LIN {X 0,Y 338.282,Z 949.56,A -85,B 0,C 180,E1 15953.701,E2 15953.701} C_VEL
LIN {X 0,Y 337.942,Z 950.503,A -85,B 0,C 180,E1 15950.977,E2 15950.977} C_VEL
LIN {X 0,Y 337.887,Z 949.725,A -85,B 0,C 180,E1 15948.28,E2 15948.28} C_VEL
LIN {X 0,Y 338.122,Z 946.903,A -85,B 0,C 180,E1 15945.416,E2 15945.416} C_VEL
LIN {X 0,Y 338.612,Z 942.779,A -85,B 0,C 180,E1 15942.968,E2 15942.968} C_VEL
LIN {X 0,Y 339.493,Z 936.406,A -85,B 0,C 180,E1 15940.349,E2 15940.349} C_VEL
LIN {X 0,Y 340.591,Z 928.995,A -85,B 0,C 180,E1 15938.1,E2 15938.1} C_VEL
LIN {X 0,Y 342.028,Z 919.535,A -85,B 0,C 180,E1 15935.872,E2 15935.872} C_VEL
LIN {X 0,Y 343.629,Z 908.396,A -85,B 0,C 180,E1 15933.837,E2 15933.837} C_VEL
LIN {X 0,Y 345.191,Z 896.567,A -85,B 0,C 180,E1 15932.124,E2 15932.124} C_VEL
LIN {X 0,Y 346.824,Z 882.835,A -85,B 0,C 180,E1 15930.578,E2 15930.578} C_VEL
LIN {X 0,Y 348.128,Z 869.607,A -85,B 0,C 180,E1 15929.424,E2 15929.424} C_VEL
LIN {X 0,Y 349.323,Z 853.76,A -85,B 0,C 180,E1 15928.401,E2 15928.401} C_VEL
LIN {X 0,Y 350.092,Z 837.915,A -85,B 0,C 180,E1 15927.713,E2 15927.713} C_VEL
LIN {X 0,Y 350.796,Z 811.808,A -85,B 0,C 180,E1 15927.074,E2 15927.074} C_VEL
LIN {X 0,Y 352.568,Z 740.463,A -85,B 0,C 180,E1 15925.552,E2 15925.552} C_VEL
LIN {X 0,Y 347.395,Z 709.374,A -85,B 0,C 180,E1 15924.417,E2 15924.417} C_VEL
LIN {X 0,Y 346.559,Z 706.204,A -85,B 0,C 180,E1 15924.151,E2 15924.151} C_VEL
LIN {X 0,Y 344.566,Z 701.019,A -85,B 0,C 180,E1 15923.183,E2 15923.183} C_VEL
LIN {X 0,Y 342.465,Z 693.939,A -85,B 0,C 180,E1 15921.676,E2 15921.676} C_VEL
LIN {X 0,Y 342.188,Z 686.245,A -85,B 0,C 180,E1 15920.292,E2 15920.292} C_VEL
LIN {X 0,Y 342.295,Z 685.366,A -85,B 0,C 180,E1 15920.142,E2 15920.142} C_VEL
LIN {X 0,Y 345.109,Z 665.644,A -85,B 0,C 180,E1 15916.768,E2 15916.768} C_VEL
LIN {X 0,Y 340.904,Z 649.05,A -85,B 0,C 180,E1 15913.12,E2 15913.12} C_VEL
LIN {X 0,Y 336.381,Z 633.612,A -85,B 0,C 180,E1 15909.442,E2 15909.442} C_VEL
LIN {X 0,Y 331.798,Z 619.998,A -85,B 0,C 180,E1 15905.935,E2 15905.935} C_VEL
LIN {X 0,Y 330.065,Z 614.784,A -85,B 0,C 180,E1 15904.435,E2 15904.435} C_VEL
LIN {X 0,Y 330.051,Z 614.615,A -85,B 0,C 180,E1 15900.009,E2 15900.009} C_VEL
LIN {X 0,Y 330.048,Z 614.676,A -85,B 0,C 180,E1 15895.703,E2 15895.703} C_VEL
LIN {X 0,Y 330.048,Z 614.671,A -85,B 0,C 180,E1 15891.386,E2 15891.386} C_VEL
LIN {X 0,Y 330.04,Z 614.659,A -85,B 0,C 180,E1 15887.151,E2 15887.151} C_VEL
LIN {X 0,Y 330.036,Z 614.677,A -85,B 0,C 180,E1 15882.848,E2 15882.848} C_VEL
LIN {X 0,Y 330.034,Z 614.681,A -85,B 0,C 180,E1 15878.589,E2 15878.589} C_VEL
LIN {X 0,Y 330.027,Z 614.651,A -85,B 0,C 180,E1 15874.198,E2 15874.198} C_VEL
LIN {X 0,Y 330.032,Z 614.688,A -85,B 0,C 180,E1 15869.792,E2 15869.792} C_VEL
LIN {X 0,Y 330.03,Z 614.644,A -85,B 0,C 180,E1 15865.467,E2 15865.467} C_VEL
LIN {X 0,Y 330.038,Z 614.685,A -85,B 0,C 180,E1 15861.132,E2 15861.132} C_VEL
LIN {X 0,Y 330.041,Z 614.643,A -85,B 0,C 180,E1 15856.727,E2 15856.727} C_VEL
LIN {X 0,Y 330.05,Z 614.68,A -85,B 0,C 180,E1 15852.421,E2 15852.421} C_VEL
LIN {X 0,Y 330.055,Z 614.642,A -85,B 0,C 180,E1 15848.011,E2 15848.011} C_VEL
LIN {X 0,Y 330.039,Z 614.678,A -85,B 0,C 180,E1 15843.648,E2 15843.648} C_VEL
LIN {X 0,Y 330.029,Z 614.653,A -85,B 0,C 180,E1 15839.306,E2 15839.306} C_VEL
LIN {X 0,Y 330.021,Z 614.678,A -85,B 0,C 180,E1 15834.96,E2 15834.96} C_VEL
LIN {X 0,Y 330.02,Z 614.672,A -85,B 0,C 180,E1 15830.76,E2 15830.76} C_VEL
LIN {X 0,Y 330.013,Z 614.663,A -85,B 0,C 180,E1 15826.509,E2 15826.509} C_VEL
LIN {X 0,Y 330.014,Z 614.69,A -85,B 0,C 180,E1 15822.182,E2 15822.182} C_VEL
LIN {X 0,Y 330.004,Z 614.675,A -85,B 0,C 180,E1 15817.933,E2 15817.933} C_VEL
LIN {X 0,Y 330.01,Z 614.666,A -85,B 0,C 180,E1 15813.553,E2 15813.553} C_VEL
LIN {X 0,Y 330.005,Z 614.672,A -85,B 0,C 180,E1 15809.371,E2 15809.371} C_VEL
LIN {X 0,Y 330.008,Z 614.675,A -85,B 0,C 180,E1 15805.194,E2 15805.194} C_VEL
LIN {X 0,Y 330.031,Z 614.845,A -85,B 0,C 180,E1 15800.976,E2 15800.976} C_VEL
LIN {X 0,Y 334.572,Z 626.543,A -85,B 0,C 180,E1 15798.208,E2 15798.208} C_VEL
LIN {X 0,Y 340.383,Z 642.032,A -85,B 0,C 180,E1 15794.934,E2 15794.934} C_VEL
LIN {X 0,Y 346.42,Z 659.693,A -85,B 0,C 180,E1 15791.594,E2 15791.594} C_VEL
LIN {X 0,Y 351.026,Z 674.252,A -85,B 0,C 180,E1 15789.066,E2 15789.066} C_VEL
LIN {X 0,Y 347.702,Z 695.465,A -85,B 0,C 180,E1 15786.551,E2 15786.551} C_VEL
LIN {X 0,Y 350.631,Z 727.811,A -85,B 0,C 180,E1 15785.557,E2 15785.557} C_VEL
LIN {X 0,Y 346.435,Z 886.846,A -85,B 0,C 180,E1 15782.34,E2 15782.34} C_VEL
LIN {X 0,Y 345.21,Z 905.278,A -85,B 0,C 180,E1 15781.685,E2 15781.685} C_VEL
LIN {X 0,Y 343.439,Z 923.152,A -85,B 0,C 180,E1 15780.753,E2 15780.753} C_VEL
LIN {X 0,Y 341.468,Z 939.767,A -85,B 0,C 180,E1 15779.582,E2 15779.582} C_VEL
LIN {X 0,Y 339.185,Z 956.678,A -85,B 0,C 180,E1 15778.046,E2 15778.046} C_VEL
LIN {X 0,Y 336.841,Z 972.419,A -85,B 0,C 180,E1 15776.25,E2 15776.25} C_VEL
LIN {X 0,Y 334.602,Z 987.176,A -85,B 0,C 180,E1 15774.167,E2 15774.167} C_VEL
LIN {X 0,Y 332.635,Z 1000.358,A -85,B 0,C 180,E1 15771.884,E2 15771.884} C_VEL
LIN {X 0,Y 331.024,Z 1012.138,A -85,B 0,C 180,E1 15769.406,E2 15769.406} C_VEL
LIN {X 0,Y 329.802,Z 1022.804,A -85,B 0,C 180,E1 15766.662,E2 15766.662} C_VEL
LIN {X 0,Y 329.096,Z 1032.024,A -85,B 0,C 180,E1 15763.709,E2 15763.709} C_VEL
LIN {X 0,Y 328.87,Z 1039.391,A -85,B 0,C 180,E1 15760.688,E2 15760.688} C_VEL
LIN {X 0,Y 329.024,Z 1044.857,A -85,B 0,C 180,E1 15757.684,E2 15757.684} C_VEL
LIN {X 0,Y 329.333,Z 1048.545,A -85,B 0,C 180,E1 15754.702,E2 15754.702} C_VEL
LIN {X 0,Y 329.583,Z 1050.525,A -85,B 0,C 180,E1 15751.739,E2 15751.739} C_VEL
LIN {X 0,Y 329.594,Z 1050.859,A -85,B 0,C 180,E1 15748.957,E2 15748.957} C_VEL
LIN {X 0,Y 329.364,Z 1049.731,A -85,B 0,C 180,E1 15746.171,E2 15746.171} C_VEL
LIN {X 0,Y 329.013,Z 1046.925,A -85,B 0,C 180,E1 15743.194,E2 15743.194} C_VEL
LIN {X 0,Y 328.773,Z 1042.425,A -85,B 0,C 180,E1 15740.177,E2 15740.177} C_VEL
LIN {X 0,Y 328.894,Z 1035.816,A -85,B 0,C 180,E1 15736.999,E2 15736.999} C_VEL
LIN {X 0,Y 329.539,Z 1027.629,A -85,B 0,C 180,E1 15733.972,E2 15733.972} C_VEL
LIN {X 0,Y 330.842,Z 1017.333,A -85,B 0,C 180,E1 15730.95,E2 15730.95} C_VEL
LIN {X 0,Y 332.674,Z 1005.885,A -85,B 0,C 180,E1 15728.234,E2 15728.234} C_VEL
LIN {X 0,Y 334.846,Z 993.661,A -85,B 0,C 180,E1 15725.853,E2 15725.853} C_VEL
LIN {X 0,Y 337.541,Z 979.122,A -85,B 0,C 180,E1 15723.525,E2 15723.525} C_VEL
LIN {X 0,Y 340.344,Z 964.071,A -85,B 0,C 180,E1 15721.581,E2 15721.581} C_VEL
LIN {X 0,Y 343.092,Z 948.032,A -85,B 0,C 180,E1 15719.917,E2 15719.917} C_VEL
LIN {X 0,Y 345.607,Z 931.814,A -85,B 0,C 180,E1 15718.589,E2 15718.589} C_VEL
LIN {X 0,Y 347.921,Z 914.248,A -85,B 0,C 180,E1 15717.493,E2 15717.493} C_VEL
LIN {X 0,Y 349.839,Z 895.574,A -85,B 0,C 180,E1 15716.67,E2 15716.67} C_VEL
LIN {X 0,Y 350.907,Z 877.121,A -85,B 0,C 180,E1 15716.145,E2 15716.145} C_VEL
LIN {X 0,Y 355.545,Z 725.644,A -85,B 0,C 180,E1 15713.02,E2 15713.02} C_VEL
LIN {X 0,Y 352.544,Z 696.426,A -85,B 0,C 180,E1 15711.908,E2 15711.908} C_VEL
LIN {X 0,Y 355.73,Z 679.777,A -85,B 0,C 180,E1 15709.864,E2 15709.864} C_VEL
LIN {X 0,Y 351.383,Z 665.481,A -85,B 0,C 180,E1 15706.928,E2 15706.928} C_VEL
LIN {X 0,Y 346.624,Z 652.331,A -85,B 0,C 180,E1 15703.812,E2 15703.812} C_VEL
LIN {X 0,Y 341.748,Z 640.208,A -85,B 0,C 180,E1 15700.475,E2 15700.475} C_VEL
LIN {X 0,Y 337.434,Z 630.747,A -85,B 0,C 180,E1 15697.404,E2 15697.404} C_VEL
LIN {X 0,Y 335.51,Z 626.722,A -85,B 0,C 180,E1 15695.95,E2 15695.95} C_VEL
LIN {X 0,Y 333.99,Z 623.294,A -85,B 0,C 180,E1 15694.666,E2 15694.666} C_VEL
LIN {X 0,Y 331.766,Z 618.774,A -85,B 0,C 180,E1 15692.772,E2 15692.772} C_VEL
LIN {X 0,Y 330.033,Z 614.822,A -85,B 0,C 180,E1 15690.923,E2 15690.923} C_VEL
LIN {X 0,Y 330.021,Z 614.671,A -85,B 0,C 180,E1 15686.835,E2 15686.835} C_VEL
LIN {X 0,Y 330.015,Z 614.669,A -85,B 0,C 180,E1 15682.63,E2 15682.63} C_VEL
LIN {X 0,Y 330.015,Z 614.666,A -85,B 0,C 180,E1 15678.366,E2 15678.366} C_VEL
LIN {X 0,Y 330.013,Z 614.663,A -85,B 0,C 180,E1 15674.182,E2 15674.182} C_VEL
LIN {X 0,Y 330.016,Z 614.663,A -85,B 0,C 180,E1 15669.944,E2 15669.944} C_VEL
LIN {X 0,Y 330.011,Z 614.668,A -85,B 0,C 180,E1 15665.563,E2 15665.563} C_VEL
LIN {X 0,Y 330.016,Z 614.674,A -85,B 0,C 180,E1 15661.117,E2 15661.117} C_VEL
LIN {X 0,Y 330.02,Z 614.683,A -85,B 0,C 180,E1 15656.873,E2 15656.873} C_VEL
LIN {X 0,Y 330.03,Z 614.685,A -85,B 0,C 180,E1 15652.514,E2 15652.514} C_VEL
LIN {X 0,Y 330.039,Z 614.681,A -85,B 0,C 180,E1 15648.107,E2 15648.107} C_VEL
LIN {X 0,Y 330.057,Z 614.851,A -85,B 0,C 180,E1 15644.088,E2 15644.088} C_VEL
LIN {X 0,Y 331.806,Z 618.825,A -85,B 0,C 180,E1 15642.099,E2 15642.099} C_VEL
LIN {X 0,Y 334.242,Z 624.749,A -85,B 0,C 180,E1 15639.512,E2 15639.512} C_VEL
LIN {X 0,Y 337.03,Z 631.317,A -85,B 0,C 180,E1 15636.878,E2 15636.878} C_VEL
LIN {X 0,Y 340.661,Z 640.852,A -85,B 0,C 180,E1 15633.504,E2 15633.504} C_VEL
LIN {X 0,Y 344.388,Z 651.989,A -85,B 0,C 180,E1 15630.041,E2 15630.041} C_VEL
LIN {X 0,Y 347.816,Z 664.12,A -85,B 0,C 180,E1 15626.697,E2 15626.697} C_VEL
LIN {X 0,Y 350.134,Z 674.513,A -85,B 0,C 180,E1 15624.117,E2 15624.117} C_VEL
LIN {X 0,Y 345.344,Z 700.754,A -85,B 0,C 180,E1 15619.464,E2 15619.464} C_VEL
LIN {X 0,Y 344.564,Z 706.075,A -85,B 0,C 180,E1 15618.576,E2 15618.576} C_VEL
LIN {X 0,Y 350.106,Z 734.115,A -85,B 0,C 180,E1 15617.096,E2 15617.096} C_VEL
LIN {X 0,Y 351.866,Z 746.069,A -85,B 0,C 180,E1 15616.573,E2 15616.573} C_VEL
LIN {X 0,Y 348.485,Z 837.417,A -85,B 0,C 180,E1 15614.49,E2 15614.49} C_VEL
LIN {X 0,Y 347.514,Z 853.648,A -85,B 0,C 180,E1 15613.812,E2 15613.812} C_VEL
LIN {X 0,Y 346.161,Z 868.356,A -85,B 0,C 180,E1 15612.908,E2 15612.908} C_VEL
LIN {X 0,Y 344.33,Z 882.931,A -85,B 0,C 180,E1 15611.68,E2 15611.68} C_VEL
LIN {X 0,Y 342.265,Z 896.285,A -85,B 0,C 180,E1 15610.211,E2 15610.211} C_VEL
LIN {X 0,Y 339.904,Z 909.258,A -85,B 0,C 180,E1 15608.365,E2 15608.365} C_VEL
LIN {X 0,Y 337.831,Z 919.497,A -85,B 0,C 180,E1 15606.504,E2 15606.504} C_VEL
LIN {X 0,Y 335.671,Z 929.228,A -85,B 0,C 180,E1 15604.261,E2 15604.261} C_VEL
LIN {X 0,Y 333.889,Z 936.762,A -85,B 0,C 180,E1 15602.008,E2 15602.008} C_VEL
LIN {X 0,Y 332.297,Z 943.342,A -85,B 0,C 180,E1 15599.37,E2 15599.37} C_VEL
LIN {X 0,Y 331.171,Z 947.855,A -85,B 0,C 180,E1 15596.734,E2 15596.734} C_VEL
LIN {X 0,Y 330.426,Z 950.744,A -85,B 0,C 180,E1 15593.921,E2 15593.921} C_VEL
LIN {X 0,Y 330.041,Z 951.708,A -85,B 0,C 180,E1 15591.078,E2 15591.078} C_VEL
LIN {X 0,Y 329.972,Z 950.962,A -85,B 0,C 180,E1 15588.369,E2 15588.369} C_VEL
LIN {X 0,Y 330.176,Z 948.422,A -85,B 0,C 180,E1 15585.635,E2 15585.635} C_VEL
LIN {X 0,Y 330.709,Z 944.112,A -85,B 0,C 180,E1 15582.928,E2 15582.928} C_VEL
LIN {X 0,Y 331.617,Z 937.787,A -85,B 0,C 180,E1 15580.247,E2 15580.247} C_VEL
LIN {X 0,Y 332.755,Z 930.471,A -85,B 0,C 180,E1 15577.945,E2 15577.945} C_VEL
LIN {X 0,Y 334.239,Z 921.09,A -85,B 0,C 180,E1 15575.665,E2 15575.665} C_VEL
LIN {X 0,Y 335.828,Z 910.621,A -85,B 0,C 180,E1 15573.67,E2 15573.67} C_VEL
LIN {X 0,Y 337.533,Z 898.355,A -85,B 0,C 180,E1 15571.819,E2 15571.819} C_VEL
LIN {X 0,Y 339.205,Z 884.971,A -85,B 0,C 180,E1 15570.253,E2 15570.253} C_VEL
LIN {X 0,Y 340.661,Z 871.088,A -85,B 0,C 180,E1 15568.991,E2 15568.991} C_VEL
LIN {X 0,Y 341.902,Z 855.452,A -85,B 0,C 180,E1 15567.947,E2 15567.947} C_VEL
LIN {X 0,Y 342.73,Z 839.818,A -85,B 0,C 180,E1 15567.23,E2 15567.23} C_VEL
LIN {X 0,Y 343.359,Z 817.533,A -85,B 0,C 180,E1 15566.648,E2 15566.648} C_VEL
LIN {X 0,Y 345.371,Z 741.623,A -85,B 0,C 180,E1 15564.998,E2 15564.998} C_VEL
LIN {X 0,Y 339.605,Z 706.444,A -85,B 0,C 180,E1 15563.661,E2 15563.661} C_VEL
LIN {X 0,Y 341.799,Z 688.88,A -85,B 0,C 180,E1 15560.741,E2 15560.741} C_VEL
LIN {X 0,Y 342.295,Z 685.366,A -85,B 0,C 180,E1 15560.142,E2 15560.142} C_VEL
LIN {X 0,Y 342.241,Z 680.167,A -85,B 0,C 180,E1 15559.178,E2 15559.178} C_VEL
LIN {X 0,Y 340.277,Z 673.413,A -85,B 0,C 180,E1 15557.717,E2 15557.717} C_VEL
LIN {X 0,Y 336.594,Z 663.57,A -85,B 0,C 180,E1 15555.441,E2 15555.441} C_VEL
LIN {X 0,Y 332.394,Z 647.593,A -85,B 0,C 180,E1 15551.769,E2 15551.769} C_VEL
LIN {X 0,Y 328.021,Z 633.059,A -85,B 0,C 180,E1 15548.168,E2 15548.168} C_VEL
LIN {X 0,Y 323.24,Z 618.973,A -85,B 0,C 180,E1 15544.338,E2 15544.338} C_VEL
LIN {X 0,Y 322.115,Z 615.767,A -85,B 0,C 180,E1 15543.305,E2 15543.305} C_VEL
LIN {X 0,Y 322.094,Z 615.599,A -85,B 0,C 180,E1 15538.957,E2 15538.957} C_VEL
LIN {X 0,Y 322.107,Z 615.676,A -85,B 0,C 180,E1 15534.516,E2 15534.516} C_VEL
LIN {X 0,Y 322.119,Z 615.677,A -85,B 0,C 180,E1 15530.019,E2 15530.019} C_VEL
LIN {X 0,Y 322.111,Z 615.657,A -85,B 0,C 180,E1 15525.557,E2 15525.557} C_VEL
LIN {X 0,Y 322.113,Z 615.639,A -85,B 0,C 180,E1 15521.153,E2 15521.153} C_VEL
LIN {X 0,Y 322.103,Z 615.673,A -85,B 0,C 180,E1 15516.786,E2 15516.786} C_VEL
LIN {X 0,Y 322.093,Z 615.649,A -85,B 0,C 180,E1 15512.396,E2 15512.396} C_VEL
LIN {X 0,Y 322.093,Z 615.659,A -85,B 0,C 180,E1 15508.155,E2 15508.155} C_VEL
LIN {X 0,Y 322.086,Z 615.662,A -85,B 0,C 180,E1 15503.682,E2 15503.682} C_VEL
LIN {X 0,Y 322.085,Z 615.647,A -85,B 0,C 180,E1 15499.313,E2 15499.313} C_VEL
LIN {X 0,Y 322.093,Z 615.661,A -85,B 0,C 180,E1 15494.931,E2 15494.931} C_VEL
LIN {X 0,Y 322.098,Z 615.644,A -85,B 0,C 180,E1 15490.554,E2 15490.554} C_VEL
LIN {X 0,Y 322.11,Z 615.658,A -85,B 0,C 180,E1 15486.237,E2 15486.237} C_VEL
LIN {X 0,Y 322.106,Z 615.637,A -85,B 0,C 180,E1 15481.735,E2 15481.735} C_VEL
LIN {X 0,Y 322.105,Z 615.67,A -85,B 0,C 180,E1 15477.51,E2 15477.51} C_VEL
LIN {X 0,Y 322.099,Z 615.636,A -85,B 0,C 180,E1 15473.226,E2 15473.226} C_VEL
LIN {X 0,Y 322.087,Z 615.677,A -85,B 0,C 180,E1 15468.806,E2 15468.806} C_VEL
LIN {X 0,Y 322.078,Z 615.652,A -85,B 0,C 180,E1 15464.516,E2 15464.516} C_VEL
LIN {X 0,Y 322.074,Z 615.655,A -85,B 0,C 180,E1 15460.162,E2 15460.162} C_VEL
LIN {X 0,Y 322.072,Z 615.676,A -85,B 0,C 180,E1 15455.809,E2 15455.809} C_VEL
LIN {X 0,Y 322.075,Z 615.68,A -85,B 0,C 180,E1 15451.44,E2 15451.44} C_VEL
LIN {X 0,Y 322.081,Z 615.679,A -85,B 0,C 180,E1 15447.094,E2 15447.094} C_VEL
LIN {X 0,Y 322.087,Z 615.675,A -85,B 0,C 180,E1 15442.747,E2 15442.747} C_VEL
LIN {X 0,Y 322.162,Z 616.103,A -85,B 0,C 180,E1 15442.008,E2 15442.008} C_VEL
LIN {X 0,Y 327.813,Z 630.366,A -85,B 0,C 180,E1 15438.558,E2 15438.558} C_VEL
LIN {X 0,Y 333.879,Z 646.764,A -85,B 0,C 180,E1 15435.03,E2 15435.03} C_VEL
LIN {X 0,Y 339.979,Z 664.942,A -85,B 0,C 180,E1 15431.542,E2 15431.542} C_VEL
LIN {X 0,Y 343.602,Z 676.825,A -85,B 0,C 180,E1 15429.449,E2 15429.449} C_VEL
LIN {X 0,Y 340.552,Z 695.511,A -85,B 0,C 180,E1 15427.185,E2 15427.185} C_VEL
LIN {X 0,Y 343.459,Z 728.591,A -85,B 0,C 180,E1 15426.135,E2 15426.135} C_VEL
LIN {X 0,Y 339.118,Z 886.31,A -85,B 0,C 180,E1 15422.886,E2 15422.886} C_VEL
LIN {X 0,Y 337.856,Z 904.729,A -85,B 0,C 180,E1 15422.22,E2 15422.22} C_VEL
LIN {X 0,Y 336.011,Z 922.754,A -85,B 0,C 180,E1 15421.26,E2 15421.26} C_VEL
LIN {X 0,Y 333.876,Z 940.037,A -85,B 0,C 180,E1 15420.008,E2 15420.008} C_VEL
LIN {X 0,Y 331.546,Z 956.6,A -85,B 0,C 180,E1 15418.457,E2 15418.457} C_VEL
LIN {X 0,Y 329.135,Z 972.132,A -85,B 0,C 180,E1 15416.63,E2 15416.63} C_VEL
LIN {X 0,Y 326.805,Z 986.777,A -85,B 0,C 180,E1 15414.492,E2 15414.492} C_VEL
LIN {X 0,Y 324.704,Z 1000.299,A -85,B 0,C 180,E1 15412.066,E2 15412.066} C_VEL
LIN {X 0,Y 323.057,Z 1011.911,A -85,B 0,C 180,E1 15409.528,E2 15409.528} C_VEL
LIN {X 0,Y 321.782,Z 1022.775,A -85,B 0,C 180,E1 15406.611,E2 15406.611} C_VEL
LIN {X 0,Y 321.114,Z 1031.499,A -85,B 0,C 180,E1 15403.689,E2 15403.689} C_VEL
LIN {X 0,Y 320.91,Z 1038.731,A -85,B 0,C 180,E1 15400.593,E2 15400.593} C_VEL
LIN {X 0,Y 321.098,Z 1044.066,A -85,B 0,C 180,E1 15397.515,E2 15397.515} C_VEL
LIN {X 0,Y 321.418,Z 1047.441,A -85,B 0,C 180,E1 15394.64,E2 15394.64} C_VEL
LIN {X 0,Y 321.671,Z 1049.298,A -85,B 0,C 180,E1 15391.782,E2 15391.782} C_VEL
LIN {X 0,Y 321.681,Z 1049.666,A -85,B 0,C 180,E1 15388.932,E2 15388.932} C_VEL
LIN {X 0,Y 321.423,Z 1048.563,A -85,B 0,C 180,E1 15386.076,E2 15386.076} C_VEL
LIN {X 0,Y 321.042,Z 1045.778,A -85,B 0,C 180,E1 15383.024,E2 15383.024} C_VEL
LIN {X 0,Y 320.792,Z 1041.326,A -85,B 0,C 180,E1 15379.948,E2 15379.948} C_VEL
LIN {X 0,Y 320.946,Z 1034.696,A -85,B 0,C 180,E1 15376.672,E2 15376.672} C_VEL
LIN {X 0,Y 321.656,Z 1026.519,A -85,B 0,C 180,E1 15373.569,E2 15373.569} C_VEL
LIN {X 0,Y 322.971,Z 1016.901,A -85,B 0,C 180,E1 15370.655,E2 15370.655} C_VEL
LIN {X 0,Y 324.984,Z 1005.117,A -85,B 0,C 180,E1 15367.764,E2 15367.764} C_VEL
LIN {X 0,Y 327.361,Z 992.635,A -85,B 0,C 180,E1 15365.264,E2 15365.264} C_VEL
LIN {X 0,Y 330.105,Z 978.696,A -85,B 0,C 180,E1 15362.978,E2 15362.978} C_VEL
LIN {X 0,Y 333.036,Z 963.853,A -85,B 0,C 180,E1 15361.003,E2 15361.003} C_VEL
LIN {X 0,Y 335.906,Z 948.039,A -85,B 0,C 180,E1 15359.314,E2 15359.314} C_VEL
LIN {X 0,Y 338.66,Z 931.126,A -85,B 0,C 180,E1 15357.898,E2 15357.898} C_VEL
LIN {X 0,Y 341.043,Z 913.911,A -85,B 0,C 180,E1 15356.804,E2 15356.804} C_VEL
LIN {X 0,Y 343.046,Z 895.285,A -85,B 0,C 180,E1 15355.965,E2 15355.965} C_VEL
LIN {X 0,Y 344.178,Z 876.781,A -85,B 0,C 180,E1 15355.425,E2 15355.425} C_VEL
LIN {X 0,Y 349.065,Z 726.518,A -85,B 0,C 180,E1 15352.264,E2 15352.264} C_VEL
LIN {X 0,Y 346.022,Z 696.479,A -85,B 0,C 180,E1 15351.079,E2 15351.079} C_VEL
LIN {X 0,Y 348.734,Z 682.628,A -85,B 0,C 180,E1 15349.331,E2 15349.331} C_VEL
LIN {X 0,Y 344.703,Z 669.207,A -85,B 0,C 180,E1 15346.482,E2 15346.482} C_VEL
LIN {X 0,Y 339.842,Z 655.593,A -85,B 0,C 180,E1 15343.143,E2 15343.143} C_VEL
LIN {X 0,Y 335.228,Z 644.252,A -85,B 0,C 180,E1 15339.886,E2 15339.886} C_VEL
LIN {X 0,Y 330.696,Z 633.649,A -85,B 0,C 180,E1 15336.342,E2 15336.342} C_VEL
LIN {X 0,Y 327.861,Z 628.133,A -85,B 0,C 180,E1 15334.134,E2 15334.134} C_VEL
LIN {X 0,Y 326.265,Z 624.54,A -85,B 0,C 180,E1 15332.64,E2 15332.64} C_VEL
LIN {X 0,Y 323.893,Z 619.847,A -85,B 0,C 180,E1 15330.415,E2 15330.415} C_VEL
LIN {X 0,Y 322.088,Z 615.8,A -85,B 0,C 180,E1 15328.2,E2 15328.2} C_VEL
LIN {X 0,Y 322.076,Z 615.654,A -85,B 0,C 180,E1 15323.801,E2 15323.801} C_VEL
LIN {X 0,Y 322.08,Z 615.654,A -85,B 0,C 180,E1 15319.589,E2 15319.589} C_VEL
LIN {X 0,Y 322.087,Z 615.656,A -85,B 0,C 180,E1 15315.299,E2 15315.299} C_VEL
LIN {X 0,Y 322.098,Z 615.66,A -85,B 0,C 180,E1 15310.915,E2 15310.915} C_VEL
LIN {X 0,Y 322.117,Z 615.669,A -85,B 0,C 180,E1 15306.595,E2 15306.595} C_VEL
LIN {X 0,Y 322.102,Z 615.677,A -85,B 0,C 180,E1 15302.134,E2 15302.134} C_VEL
LIN {X 0,Y 322.099,Z 615.67,A -85,B 0,C 180,E1 15297.865,E2 15297.865} C_VEL
LIN {X 0,Y 322.088,Z 615.668,A -85,B 0,C 180,E1 15293.402,E2 15293.402} C_VEL
LIN {X 0,Y 322.086,Z 615.668,A -85,B 0,C 180,E1 15289.084,E2 15289.084} C_VEL
LIN {X 0,Y 322.132,Z 616.005,A -85,B 0,C 180,E1 15286.63,E2 15286.63} C_VEL
LIN {X 0,Y 324.448,Z 621.314,A -85,B 0,C 180,E1 15283.713,E2 15283.713} C_VEL
LIN {X 0,Y 326.371,Z 625.626,A -85,B 0,C 180,E1 15281.606,E2 15281.606} C_VEL
LIN {X 0,Y 328.211,Z 629.924,A -85,B 0,C 180,E1 15279.678,E2 15279.678} C_VEL
LIN {X 0,Y 331.031,Z 636.814,A -85,B 0,C 180,E1 15276.88,E2 15276.88} C_VEL
LIN {X 0,Y 334.3,Z 645.526,A -85,B 0,C 180,E1 15273.726,E2 15273.726} C_VEL
LIN {X 0,Y 337.901,Z 656.63,A -85,B 0,C 180,E1 15270.19,E2 15270.19} C_VEL
LIN {X 0,Y 341.08,Z 668.141,A -85,B 0,C 180,E1 15266.958,E2 15266.958} C_VEL
LIN {X 0,Y 343.152,Z 677.532,A -85,B 0,C 180,E1 15264.56,E2 15264.56} C_VEL
LIN {X 0,Y 338.173,Z 703.553,A -85,B 0,C 180,E1 15259.868,E2 15259.868} C_VEL
LIN {X 0,Y 337.894,Z 706.302,A -85,B 0,C 180,E1 15259.451,E2 15259.451} C_VEL
LIN {X 0,Y 343.67,Z 735.552,A -85,B 0,C 180,E1 15257.866,E2 15257.866} C_VEL
LIN {X 0,Y 345.402,Z 747.206,A -85,B 0,C 180,E1 15257.334,E2 15257.334} C_VEL
LIN {X 0,Y 341.868,Z 838.036,A -85,B 0,C 180,E1 15255.23,E2 15255.23} C_VEL
LIN {X 0,Y 340.84,Z 854.294,A -85,B 0,C 180,E1 15254.54,E2 15254.54} C_VEL
LIN {X 0,Y 339.356,Z 869.483,A -85,B 0,C 180,E1 15253.586,E2 15253.586} C_VEL
LIN {X 0,Y 337.349,Z 884.526,A -85,B 0,C 180,E1 15252.283,E2 15252.283} C_VEL
LIN {X 0,Y 335.172,Z 897.677,A -85,B 0,C 180,E1 15250.791,E2 15250.791} C_VEL
LIN {X 0,Y 332.687,Z 910.556,A -85,B 0,C 180,E1 15248.912,E2 15248.912} C_VEL
LIN {X 0,Y 330.291,Z 921.628,A -85,B 0,C 180,E1 15246.826,E2 15246.826} C_VEL
LIN {X 0,Y 328.04,Z 931.147,A -85,B 0,C 180,E1 15244.536,E2 15244.536} C_VEL
LIN {X 0,Y 326.036,Z 939.016,A -85,B 0,C 180,E1 15242.042,E2 15242.042} C_VEL
LIN {X 0,Y 324.506,Z 944.917,A -85,B 0,C 180,E1 15239.537,E2 15239.537} C_VEL
LIN {X 0,Y 323.247,Z 949.563,A -85,B 0,C 180,E1 15236.628,E2 15236.628} C_VEL
LIN {X 0,Y 322.511,Z 952.107,A -85,B 0,C 180,E1 15233.854,E2 15233.854} C_VEL
LIN {X 0,Y 322.119,Z 952.926,A -85,B 0,C 180,E1 15230.882,E2 15230.882} C_VEL
LIN {X 0,Y 322.062,Z 951.937,A -85,B 0,C 180,E1 15228.086,E2 15228.086} C_VEL
LIN {X 0,Y 322.313,Z 949.186,A -85,B 0,C 180,E1 15225.253,E2 15225.253} C_VEL
LIN {X 0,Y 322.898,Z 944.675,A -85,B 0,C 180,E1 15222.518,E2 15222.518} C_VEL
LIN {X 0,Y 323.822,Z 938.62,A -85,B 0,C 180,E1 15219.943,E2 15219.943} C_VEL
LIN {X 0,Y 325.019,Z 931.247,A -85,B 0,C 180,E1 15217.601,E2 15217.601} C_VEL
LIN {X 0,Y 326.583,Z 921.799,A -85,B 0,C 180,E1 15215.27,E2 15215.27} C_VEL
LIN {X 0,Y 328.327,Z 910.715,A -85,B 0,C 180,E1 15213.142,E2 15213.142} C_VEL
LIN {X 0,Y 330.046,Z 898.834,A -85,B 0,C 180,E1 15211.333,E2 15211.333} C_VEL
LIN {X 0,Y 331.787,Z 885.386,A -85,B 0,C 180,E1 15209.741,E2 15209.741} C_VEL
LIN {X 0,Y 333.304,Z 871.356,A -85,B 0,C 180,E1 15208.453,E2 15208.453} C_VEL
LIN {X 0,Y 334.6,Z 855.565,A -85,B 0,C 180,E1 15207.388,E2 15207.388} C_VEL
LIN {X 0,Y 335.447,Z 839.861,A -85,B 0,C 180,E1 15206.668,E2 15206.668} C_VEL
LIN {X 0,Y 336.137,Z 816.358,A -85,B 0,C 180,E1 15206.053,E2 15206.053} C_VEL
LIN {X 0,Y 338.188,Z 742.721,A -85,B 0,C 180,E1 15204.422,E2 15204.422} C_VEL
LIN {X 0,Y 332.289,Z 706.332,A -85,B 0,C 180,E1 15203,E2 15203} C_VEL
LIN {X 0,Y 333.364,Z 697.56,A -85,B 0,C 180,E1 15201.548,E2 15201.548} C_VEL
LIN {X 0,Y 337.399,Z 670.235,A -85,B 0,C 180,E1 15196.809,E2 15196.809} C_VEL
LIN {X 0,Y 337.527,Z 667.454,A -85,B 0,C 180,E1 15196.291,E2 15196.291} C_VEL
LIN {X 0,Y 336.594,Z 663.57,A -85,B 0,C 180,E1 15195.441,E2 15195.441} C_VEL
LIN {X 0,Y 334.538,Z 659.376,A -85,B 0,C 180,E1 15194.383,E2 15194.383} C_VEL
LIN {X 0,Y 325.4,Z 649.582,A -85,B 0,C 180,E1 15191.255,E2 15191.255} C_VEL
LIN {X 0,Y 324.049,Z 646.601,A -85,B 0,C 180,E1 15190.454,E2 15190.454} C_VEL
LIN {X 0,Y 319.525,Z 632.114,A -85,B 0,C 180,E1 15186.681,E2 15186.681} C_VEL
LIN {X 0,Y 315.121,Z 619.584,A -85,B 0,C 180,E1 15183.075,E2 15183.075} C_VEL
LIN {X 0,Y 314.193,Z 616.761,A -85,B 0,C 180,E1 15182.165,E2 15182.165} C_VEL
LIN {X 0,Y 314.164,Z 616.594,A -85,B 0,C 180,E1 15177.842,E2 15177.842} C_VEL
LIN {X 0,Y 314.166,Z 616.649,A -85,B 0,C 180,E1 15173.476,E2 15173.476} C_VEL
LIN {X 0,Y 314.162,Z 616.658,A -85,B 0,C 180,E1 15168.963,E2 15168.963} C_VEL
LIN {X 0,Y 314.161,Z 616.663,A -85,B 0,C 180,E1 15164.442,E2 15164.442} C_VEL
LIN {X 0,Y 314.166,Z 616.632,A -85,B 0,C 180,E1 15159.914,E2 15159.914} C_VEL
LIN {X 0,Y 314.169,Z 616.64,A -85,B 0,C 180,E1 15155.438,E2 15155.438} C_VEL
LIN {X 0,Y 314.181,Z 616.655,A -85,B 0,C 180,E1 15151.035,E2 15151.035} C_VEL
LIN {X 0,Y 314.166,Z 616.62,A -85,B 0,C 180,E1 15146.579,E2 15146.579} C_VEL
LIN {X 0,Y 314.156,Z 616.663,A -85,B 0,C 180,E1 15142.059,E2 15142.059} C_VEL
LIN {X 0,Y 314.142,Z 616.617,A -85,B 0,C 180,E1 15137.6,E2 15137.6} C_VEL
LIN {X 0,Y 314.147,Z 616.666,A -85,B 0,C 180,E1 15133.109,E2 15133.109} C_VEL
LIN {X 0,Y 314.152,Z 616.616,A -85,B 0,C 180,E1 15128.603,E2 15128.603} C_VEL
LIN {X 0,Y 314.163,Z 616.66,A -85,B 0,C 180,E1 15124.198,E2 15124.198} C_VEL
LIN {X 0,Y 314.173,Z 616.621,A -85,B 0,C 180,E1 15119.636,E2 15119.636} C_VEL
LIN {X 0,Y 314.158,Z 616.657,A -85,B 0,C 180,E1 15115.254,E2 15115.254} C_VEL
LIN {X 0,Y 314.146,Z 616.644,A -85,B 0,C 180,E1 15110.843,E2 15110.843} C_VEL
LIN {X 0,Y 314.131,Z 616.638,A -85,B 0,C 180,E1 15106.377,E2 15106.377} C_VEL
LIN {X 0,Y 314.138,Z 616.667,A -85,B 0,C 180,E1 15101.825,E2 15101.825} C_VEL
LIN {X 0,Y 314.135,Z 616.656,A -85,B 0,C 180,E1 15097.546,E2 15097.546} C_VEL
LIN {X 0,Y 314.151,Z 616.643,A -85,B 0,C 180,E1 15093.132,E2 15093.132} C_VEL
LIN {X 0,Y 314.165,Z 616.644,A -85,B 0,C 180,E1 15088.751,E2 15088.751} C_VEL
LIN {X 0,Y 314.161,Z 616.651,A -85,B 0,C 180,E1 15084.251,E2 15084.251} C_VEL
LIN {X 0,Y 314.191,Z 617.076,A -85,B 0,C 180,E1 15083.229,E2 15083.229} C_VEL
LIN {X 0,Y 319.821,Z 630.963,A -85,B 0,C 180,E1 15079.674,E2 15079.674} C_VEL
LIN {X 0,Y 325.933,Z 647.385,A -85,B 0,C 180,E1 15075.987,E2 15075.987} C_VEL
LIN {X 0,Y 331.742,Z 664.66,A -85,B 0,C 180,E1 15072.518,E2 15072.518} C_VEL
LIN {X 0,Y 336.242,Z 679.007,A -85,B 0,C 180,E1 15069.897,E2 15069.897} C_VEL
LIN {X 0,Y 333.42,Z 695.85,A -85,B 0,C 180,E1 15067.82,E2 15067.82} C_VEL
LIN {X 0,Y 336.325,Z 729.344,A -85,B 0,C 180,E1 15066.738,E2 15066.738} C_VEL
LIN {X 0,Y 331.822,Z 885.719,A -85,B 0,C 180,E1 15063.454,E2 15063.454} C_VEL
LIN {X 0,Y 330.516,Z 904.15,A -85,B 0,C 180,E1 15062.772,E2 15062.772} C_VEL
LIN {X 0,Y 328.564,Z 922.565,A -85,B 0,C 180,E1 15061.767,E2 15061.767} C_VEL
LIN {X 0,Y 326.356,Z 939.733,A -85,B 0,C 180,E1 15060.489,E2 15060.489} C_VEL
LIN {X 0,Y 323.922,Z 956.374,A -85,B 0,C 180,E1 15058.887,E2 15058.887} C_VEL
LIN {X 0,Y 321.424,Z 971.856,A -85,B 0,C 180,E1 15057.012,E2 15057.012} C_VEL
LIN {X 0,Y 319.018,Z 986.343,A -85,B 0,C 180,E1 15054.834,E2 15054.834} C_VEL
LIN {X 0,Y 316.893,Z 999.494,A -85,B 0,C 180,E1 15052.412,E2 15052.412} C_VEL
LIN {X 0,Y 315.092,Z 1011.683,A -85,B 0,C 180,E1 15049.656,E2 15049.656} C_VEL
LIN {X 0,Y 313.859,Z 1021.78,A -85,B 0,C 180,E1 15046.852,E2 15046.852} C_VEL
LIN {X 0,Y 313.159,Z 1030.481,A -85,B 0,C 180,E1 15043.855,E2 15043.855} C_VEL
LIN {X 0,Y 312.951,Z 1037.686,A -85,B 0,C 180,E1 15040.679,E2 15040.679} C_VEL
LIN {X 0,Y 313.158,Z 1042.989,A -85,B 0,C 180,E1 15037.522,E2 15037.522} C_VEL
LIN {X 0,Y 313.504,Z 1046.327,A -85,B 0,C 180,E1 15034.574,E2 15034.574} C_VEL
LIN {X 0,Y 313.769,Z 1048.136,A -85,B 0,C 180,E1 15031.644,E2 15031.644} C_VEL
LIN {X 0,Y 313.757,Z 1048.442,A -85,B 0,C 180,E1 15028.722,E2 15028.722} C_VEL
LIN {X 0,Y 313.455,Z 1047.265,A -85,B 0,C 180,E1 15025.793,E2 15025.793} C_VEL
LIN {X 0,Y 313.048,Z 1044.399,A -85,B 0,C 180,E1 15022.66,E2 15022.66} C_VEL
LIN {X 0,Y 312.807,Z 1039.86,A -85,B 0,C 180,E1 15019.503,E2 15019.503} C_VEL
LIN {X 0,Y 313.033,Z 1033.137,A -85,B 0,C 180,E1 15016.14,E2 15016.14} C_VEL
LIN {X 0,Y 313.893,Z 1024.587,A -85,B 0,C 180,E1 15012.863,E2 15012.863} C_VEL
LIN {X 0,Y 315.485,Z 1014.31,A -85,B 0,C 180,E1 15009.735,E2 15009.735} C_VEL
LIN {X 0,Y 317.704,Z 1002.481,A -85,B 0,C 180,E1 15006.834,E2 15006.834} C_VEL
LIN {X 0,Y 320.425,Z 989.173,A -85,B 0,C 180,E1 15004.196,E2 15004.196} C_VEL
LIN {X 0,Y 323.337,Z 975.295,A -85,B 0,C 180,E1 15001.964,E2 15001.964} C_VEL
LIN {X 0,Y 326.35,Z 960.581,A -85,B 0,C 180,E1 15000.04,E2 15000.04} C_VEL
LIN {X 0,Y 329.431,Z 944.189,A -85,B 0,C 180,E1 14998.327,E2 14998.327} C_VEL
LIN {X 0,Y 332.352,Z 926.698,A -85,B 0,C 180,E1 14996.905,E2 14996.905} C_VEL
LIN {X 0,Y 334.821,Z 909.191,A -85,B 0,C 180,E1 14995.846,E2 14995.846} C_VEL
LIN {X 0,Y 336.72,Z 890.808,A -85,B 0,C 180,E1 14995.066,E2 14995.066} C_VEL
LIN {X 0,Y 337.747,Z 871.011,A -85,B 0,C 180,E1 14994.546,E2 14994.546} C_VEL
LIN {X 0,Y 342.665,Z 727.468,A -85,B 0,C 180,E1 14991.479,E2 14991.479} C_VEL
LIN {X 0,Y 339.64,Z 697.148,A -85,B 0,C 180,E1 14990.245,E2 14990.245} C_VEL
LIN {X 0,Y 340.033,Z 694.015,A -85,B 0,C 180,E1 14989.912,E2 14989.912} C_VEL
LIN {X 0,Y 341.863,Z 685.853,A -85,B 0,C 180,E1 14988.848,E2 14988.848} C_VEL
LIN {X 0,Y 337.934,Z 672.66,A -85,B 0,C 180,E1 14985.949,E2 14985.949} C_VEL
LIN {X 0,Y 333.389,Z 659.694,A -85,B 0,C 180,E1 14982.671,E2 14982.671} C_VEL
LIN {X 0,Y 329.241,Z 649.345,A -85,B 0,C 180,E1 14979.623,E2 14979.623} C_VEL
LIN {X 0,Y 324.9,Z 639.042,A -85,B 0,C 180,E1 14976.109,E2 14976.109} C_VEL
LIN {X 0,Y 322.262,Z 633.75,A -85,B 0,C 180,E1 14973.95,E2 14973.95} C_VEL
LIN {X 0,Y 320.66,Z 630.168,A -85,B 0,C 180,E1 14972.433,E2 14972.433} C_VEL
LIN {X 0,Y 318.323,Z 625.502,A -85,B 0,C 180,E1 14970.169,E2 14970.169} C_VEL
LIN {X 0,Y 316.051,Z 620.912,A -85,B 0,C 180,E1 14967.649,E2 14967.649} C_VEL
LIN {X 0,Y 314.272,Z 617.305,A -85,B 0,C 180,E1 14965.372,E2 14965.372} C_VEL
LIN {X 0,Y 314.136,Z 616.685,A -85,B 0,C 180,E1 14964.453,E2 14964.453} C_VEL
LIN {X 0,Y 314.132,Z 616.646,A -85,B 0,C 180,E1 14959.911,E2 14959.911} C_VEL
LIN {X 0,Y 314.139,Z 616.647,A -85,B 0,C 180,E1 14955.507,E2 14955.507} C_VEL
LIN {X 0,Y 314.147,Z 616.655,A -85,B 0,C 180,E1 14951.195,E2 14951.195} C_VEL
LIN {X 0,Y 314.167,Z 616.662,A -85,B 0,C 180,E1 14946.762,E2 14946.762} C_VEL
LIN {X 0,Y 314.164,Z 616.666,A -85,B 0,C 180,E1 14942.188,E2 14942.188} C_VEL
LIN {X 0,Y 314.157,Z 616.66,A -85,B 0,C 180,E1 14937.811,E2 14937.811} C_VEL
LIN {X 0,Y 314.15,Z 616.656,A -85,B 0,C 180,E1 14933.42,E2 14933.42} C_VEL
LIN {X 0,Y 314.209,Z 616.929,A -85,B 0,C 180,E1 14929.839,E2 14929.839} C_VEL
LIN {X 0,Y 315.995,Z 620.859,A -85,B 0,C 180,E1 14927.203,E2 14927.203} C_VEL
LIN {X 0,Y 318.561,Z 626.542,A -85,B 0,C 180,E1 14923.966,E2 14923.966} C_VEL
LIN {X 0,Y 320.406,Z 630.824,A -85,B 0,C 180,E1 14921.816,E2 14921.816} C_VEL
LIN {X 0,Y 322.36,Z 635.535,A -85,B 0,C 180,E1 14919.672,E2 14919.672} C_VEL
LIN {X 0,Y 325.686,Z 643.75,A -85,B 0,C 180,E1 14916.286,E2 14916.286} C_VEL
LIN {X 0,Y 329.184,Z 653.916,A -85,B 0,C 180,E1 14912.7,E2 14912.7} C_VEL
LIN {X 0,Y 332.518,Z 664.969,A -85,B 0,C 180,E1 14909.257,E2 14909.257} C_VEL
LIN {X 0,Y 335.476,Z 677.081,A -85,B 0,C 180,E1 14905.922,E2 14905.922} C_VEL
LIN {X 0,Y 336.137,Z 680.911,A -85,B 0,C 180,E1 14904.964,E2 14904.964} C_VEL
LIN {X 0,Y 331.271,Z 705.81,A -85,B 0,C 180,E1 14900.442,E2 14900.442} C_VEL
LIN {X 0,Y 336.729,Z 733.763,A -85,B 0,C 180,E1 14898.832,E2 14898.832} C_VEL
LIN {X 0,Y 338.993,Z 748.504,A -85,B 0,C 180,E1 14898.122,E2 14898.122} C_VEL
LIN {X 0,Y 335.311,Z 838.717,A -85,B 0,C 180,E1 14895.997,E2 14895.997} C_VEL
LIN {X 0,Y 334.23,Z 854.995,A -85,B 0,C 180,E1 14895.295,E2 14895.295} C_VEL
LIN {X 0,Y 332.678,Z 870.157,A -85,B 0,C 180,E1 14894.331,E2 14894.331} C_VEL
LIN {X 0,Y 330.56,Z 885.253,A -85,B 0,C 180,E1 14893.006,E2 14893.006} C_VEL
LIN {X 0,Y 328.409,Z 897.744,A -85,B 0,C 180,E1 14891.584,E2 14891.584} C_VEL
LIN {X 0,Y 325.76,Z 910.769,A -85,B 0,C 180,E1 14889.674,E2 14889.674} C_VEL
LIN {X 0,Y 323.32,Z 921.523,A -85,B 0,C 180,E1 14887.657,E2 14887.657} C_VEL
LIN {X 0,Y 320.777,Z 931.664,A -85,B 0,C 180,E1 14885.215,E2 14885.215} C_VEL
LIN {X 0,Y 318.686,Z 939.391,A -85,B 0,C 180,E1 14882.771,E2 14882.771} C_VEL
LIN {X 0,Y 316.93,Z 945.7,A -85,B 0,C 180,E1 14880.107,E2 14880.107} C_VEL
LIN {X 0,Y 315.619,Z 950.219,A -85,B 0,C 180,E1 14877.345,E2 14877.345} C_VEL
LIN {X 0,Y 314.728,Z 953.121,A -85,B 0,C 180,E1 14874.393,E2 14874.393} C_VEL
LIN {X 0,Y 314.256,Z 954.12,A -85,B 0,C 180,E1 14871.462,E2 14871.462} C_VEL
LIN {X 0,Y 314.14,Z 953.367,A -85,B 0,C 180,E1 14868.469,E2 14868.469} C_VEL
LIN {X 0,Y 314.362,Z 950.691,A -85,B 0,C 180,E1 14865.479,E2 14865.479} C_VEL
LIN {X 0,Y 314.943,Z 946.354,A -85,B 0,C 180,E1 14862.653,E2 14862.653} C_VEL
LIN {X 0,Y 315.939,Z 940.003,A -85,B 0,C 180,E1 14859.84,E2 14859.84} C_VEL
LIN {X 0,Y 317.185,Z 932.678,A -85,B 0,C 180,E1 14857.426,E2 14857.426} C_VEL
LIN {X 0,Y 318.801,Z 923.301,A -85,B 0,C 180,E1 14855.038,E2 14855.038} C_VEL
LIN {X 0,Y 320.53,Z 912.876,A -85,B 0,C 180,E1 14852.95,E2 14852.95} C_VEL
LIN {X 0,Y 322.401,Z 900.521,A -85,B 0,C 180,E1 14850.995,E2 14850.995} C_VEL
LIN {X 0,Y 324.19,Z 887.438,A -85,B 0,C 180,E1 14849.381,E2 14849.381} C_VEL
LIN {X 0,Y 325.873,Z 872.726,A -85,B 0,C 180,E1 14847.978,E2 14847.978} C_VEL
LIN {X 0,Y 327.221,Z 857.13,A -85,B 0,C 180,E1 14846.891,E2 14846.891} C_VEL
LIN {X 0,Y 328.138,Z 841.411,A -85,B 0,C 180,E1 14846.134,E2 14846.134} C_VEL
LIN {X 0,Y 328.811,Z 819.588,A -85,B 0,C 180,E1 14845.533,E2 14845.533} C_VEL
LIN {X 0,Y 331.02,Z 743.715,A -85,B 0,C 180,E1 14843.817,E2 14843.817} C_VEL
LIN {X 0,Y 324.987,Z 705.67,A -85,B 0,C 180,E1 14842.264,E2 14842.264} C_VEL
LIN {X 0,Y 329.152,Z 677.77,A -85,B 0,C 180,E1 14837.366,E2 14837.366} C_VEL
LIN {X 0,Y 330.241,Z 670.505,A -85,B 0,C 180,E1 14836.072,E2 14836.072} C_VEL
LIN {X 0,Y 326.198,Z 654.3,A -85,B 0,C 180,E1 14832.334,E2 14832.334} C_VEL
LIN {X 0,Y 324.049,Z 646.601,A -85,B 0,C 180,E1 14830.454,E2 14830.454} C_VEL
LIN {X 0,Y 322.313,Z 643.196,A -85,B 0,C 180,E1 14829.49,E2 14829.49} C_VEL
LIN {X 0,Y 317.644,Z 638.786,A -85,B 0,C 180,E1 14827.852,E2 14827.852} C_VEL
LIN {X 0,Y 312.522,Z 634.059,A -85,B 0,C 180,E1 14825.987,E2 14825.987} C_VEL
LIN {X 0,Y 311.069,Z 631.353,A -85,B 0,C 180,E1 14825.126,E2 14825.126} C_VEL
LIN {X 0,Y 307.113,Z 620.399,A -85,B 0,C 180,E1 14821.831,E2 14821.831} C_VEL
LIN {X 0,Y 306.24,Z 617.707,A -85,B 0,C 180,E1 14820.89,E2 14820.89} C_VEL
LIN {X 0,Y 306.231,Z 617.613,A -85,B 0,C 180,E1 14816.366,E2 14816.366} C_VEL
LIN {X 0,Y 306.237,Z 617.63,A -85,B 0,C 180,E1 14811.894,E2 14811.894} C_VEL
LIN {X 0,Y 306.23,Z 617.624,A -85,B 0,C 180,E1 14807.478,E2 14807.478} C_VEL
LIN {X 0,Y 306.224,Z 617.643,A -85,B 0,C 180,E1 14802.996,E2 14802.996} C_VEL
LIN {X 0,Y 306.218,Z 617.645,A -85,B 0,C 180,E1 14798.584,E2 14798.584} C_VEL
LIN {X 0,Y 306.212,Z 617.614,A -85,B 0,C 180,E1 14794.169,E2 14794.169} C_VEL
LIN {X 0,Y 306.218,Z 617.655,A -85,B 0,C 180,E1 14789.709,E2 14789.709} C_VEL
LIN {X 0,Y 306.22,Z 617.608,A -85,B 0,C 180,E1 14785.249,E2 14785.249} C_VEL
LIN {X 0,Y 306.236,Z 617.645,A -85,B 0,C 180,E1 14780.848,E2 14780.848} C_VEL
LIN {X 0,Y 306.231,Z 617.61,A -85,B 0,C 180,E1 14776.273,E2 14776.273} C_VEL
LIN {X 0,Y 306.22,Z 617.645,A -85,B 0,C 180,E1 14771.871,E2 14771.871} C_VEL
LIN {X 0,Y 306.205,Z 617.618,A -85,B 0,C 180,E1 14767.317,E2 14767.317} C_VEL
LIN {X 0,Y 306.202,Z 617.633,A -85,B 0,C 180,E1 14762.808,E2 14762.808} C_VEL
LIN {X 0,Y 306.205,Z 617.637,A -85,B 0,C 180,E1 14758.316,E2 14758.316} C_VEL
LIN {X 0,Y 306.222,Z 617.617,A -85,B 0,C 180,E1 14753.815,E2 14753.815} C_VEL
LIN {X 0,Y 306.227,Z 617.654,A -85,B 0,C 180,E1 14749.274,E2 14749.274} C_VEL
LIN {X 0,Y 306.218,Z 617.621,A -85,B 0,C 180,E1 14744.858,E2 14744.858} C_VEL
LIN {X 0,Y 306.202,Z 617.633,A -85,B 0,C 180,E1 14740.347,E2 14740.347} C_VEL
LIN {X 0,Y 306.195,Z 617.654,A -85,B 0,C 180,E1 14735.91,E2 14735.91} C_VEL
LIN {X 0,Y 306.199,Z 617.658,A -85,B 0,C 180,E1 14731.45,E2 14731.45} C_VEL
LIN {X 0,Y 306.209,Z 617.657,A -85,B 0,C 180,E1 14726.955,E2 14726.955} C_VEL
LIN {X 0,Y 306.264,Z 617.932,A -85,B 0,C 180,E1 14724.554,E2 14724.554} C_VEL
LIN {X 0,Y 311.867,Z 631.715,A -85,B 0,C 180,E1 14720.833,E2 14720.833} C_VEL
LIN {X 0,Y 317.813,Z 647.653,A -85,B 0,C 180,E1 14717.069,E2 14717.069} C_VEL
LIN {X 0,Y 323.688,Z 664.872,A -85,B 0,C 180,E1 14713.456,E2 14713.456} C_VEL
LIN {X 0,Y 328.825,Z 681.616,A -85,B 0,C 180,E1 14710.293,E2 14710.293} C_VEL
LIN {X 0,Y 326.323,Z 695.934,A -85,B 0,C 180,E1 14708.495,E2 14708.495} C_VEL
LIN {X 0,Y 329.225,Z 730.19,A -85,B 0,C 180,E1 14707.365,E2 14707.365} C_VEL
LIN {X 0,Y 324.557,Z 885.162,A -85,B 0,C 180,E1 14704.045,E2 14704.045} C_VEL
LIN {X 0,Y 323.218,Z 903.472,A -85,B 0,C 180,E1 14703.355,E2 14703.355} C_VEL
LIN {X 0,Y 321.19,Z 922.008,A -85,B 0,C 180,E1 14702.321,E2 14702.321} C_VEL
LIN {X 0,Y 318.89,Z 939.207,A -85,B 0,C 180,E1 14701.01,E2 14701.01} C_VEL
LIN {X 0,Y 316.448,Z 955.284,A -85,B 0,C 180,E1 14699.428,E2 14699.428} C_VEL
LIN {X 0,Y 313.85,Z 970.805,A -85,B 0,C 180,E1 14697.513,E2 14697.513} C_VEL
LIN {X 0,Y 311.335,Z 985.302,A -85,B 0,C 180,E1 14695.286,E2 14695.286} C_VEL
LIN {X 0,Y 309.116,Z 998.482,A -85,B 0,C 180,E1 14692.802,E2 14692.802} C_VEL
LIN {X 0,Y 307.234,Z 1010.674,A -85,B 0,C 180,E1 14689.982,E2 14689.982} C_VEL
LIN {X 0,Y 305.94,Z 1020.778,A -85,B 0,C 180,E1 14687.106,E2 14687.106} C_VEL
LIN {X 0,Y 305.205,Z 1029.461,A -85,B 0,C 180,E1 14684.03,E2 14684.03} C_VEL
LIN {X 0,Y 304.99,Z 1036.64,A -85,B 0,C 180,E1 14680.77,E2 14680.77} C_VEL
LIN {X 0,Y 305.218,Z 1041.912,A -85,B 0,C 180,E1 14677.53,E2 14677.53} C_VEL
LIN {X 0,Y 305.591,Z 1045.211,A -85,B 0,C 180,E1 14674.504,E2 14674.504} C_VEL
LIN {X 0,Y 305.867,Z 1046.972,A -85,B 0,C 180,E1 14671.499,E2 14671.499} C_VEL
LIN {X 0,Y 305.842,Z 1047.25,A -85,B 0,C 180,E1 14668.689,E2 14668.689} C_VEL
LIN {X 0,Y 305.51,Z 1046.099,A -85,B 0,C 180,E1 14665.683,E2 14665.683} C_VEL
LIN {X 0,Y 305.071,Z 1043.252,A -85,B 0,C 180,E1 14662.467,E2 14662.467} C_VEL
LIN {X 0,Y 304.826,Z 1038.728,A -85,B 0,C 180,E1 14659.225,E2 14659.225} C_VEL
LIN {X 0,Y 305.097,Z 1032.038,A -85,B 0,C 180,E1 14655.772,E2 14655.772} C_VEL
LIN {X 0,Y 306.011,Z 1023.803,A -85,B 0,C 180,E1 14652.507,E2 14652.507} C_VEL
LIN {X 0,Y 307.739,Z 1013.459,A -85,B 0,C 180,E1 14649.259,E2 14649.259} C_VEL
LIN {X 0,Y 310.084,Z 1001.783,A -85,B 0,C 180,E1 14646.312,E2 14646.312} C_VEL
LIN {X 0,Y 312.937,Z 988.685,A -85,B 0,C 180,E1 14643.633,E2 14643.633} C_VEL
LIN {X 0,Y 316.136,Z 974.318,A -85,B 0,C 180,E1 14641.267,E2 14641.267} C_VEL
LIN {X 0,Y 319.463,Z 958.915,A -85,B 0,C 180,E1 14639.221,E2 14639.221} C_VEL
LIN {X 0,Y 322.717,Z 942.426,A -85,B 0,C 180,E1 14637.483,E2 14637.483} C_VEL
LIN {X 0,Y 325.686,Z 925.417,A -85,B 0,C 180,E1 14636.095,E2 14636.095} C_VEL
LIN {X 0,Y 328.183,Z 908.369,A -85,B 0,C 180,E1 14635.057,E2 14635.057} C_VEL
LIN {X 0,Y 330.152,Z 889.98,A -85,B 0,C 180,E1 14634.268,E2 14634.268} C_VEL
LIN {X 0,Y 331.218,Z 870.166,A -85,B 0,C 180,E1 14633.741,E2 14633.741} C_VEL
LIN {X 0,Y 336.342,Z 728.413,A -85,B 0,C 180,E1 14630.662,E2 14630.662} C_VEL
LIN {X 0,Y 333.41,Z 698.451,A -85,B 0,C 180,E1 14629.41,E2 14629.41} C_VEL
LIN {X 0,Y 333.439,Z 695.448,A -85,B 0,C 180,E1 14629.179,E2 14629.179} C_VEL
LIN {X 0,Y 334.935,Z 688.719,A -85,B 0,C 180,E1 14628.264,E2 14628.264} C_VEL
LIN {X 0,Y 330.852,Z 674.968,A -85,B 0,C 180,E1 14625.127,E2 14625.127} C_VEL
LIN {X 0,Y 326.535,Z 662.734,A -85,B 0,C 180,E1 14621.876,E2 14621.876} C_VEL
LIN {X 0,Y 322.084,Z 651.412,A -85,B 0,C 180,E1 14618.379,E2 14618.379} C_VEL
LIN {X 0,Y 318.257,Z 642.906,A -85,B 0,C 180,E1 14615.231,E2 14615.231} C_VEL
LIN {X 0,Y 316.411,Z 638.921,A -85,B 0,C 180,E1 14613.573,E2 14613.573} C_VEL
LIN {X 0,Y 314.801,Z 635.384,A -85,B 0,C 180,E1 14612.002,E2 14612.002} C_VEL
LIN {X 0,Y 312.861,Z 631.28,A -85,B 0,C 180,E1 14609.994,E2 14609.994} C_VEL
LIN {X 0,Y 310.578,Z 626.655,A -85,B 0,C 180,E1 14607.41,E2 14607.41} C_VEL
LIN {X 0,Y 308.39,Z 622.259,A -85,B 0,C 180,E1 14604.519,E2 14604.519} C_VEL
LIN {X 0,Y 306.229,Z 617.771,A -85,B 0,C 180,E1 14600.715,E2 14600.715} C_VEL
LIN {X 0,Y 306.199,Z 617.649,A -85,B 0,C 180,E1 14596.255,E2 14596.255} C_VEL
LIN {X 0,Y 306.197,Z 617.659,A -85,B 0,C 180,E1 14591.871,E2 14591.871} C_VEL
LIN {X 0,Y 306.201,Z 617.652,A -85,B 0,C 180,E1 14587.316,E2 14587.316} C_VEL
LIN {X 0,Y 306.212,Z 617.643,A -85,B 0,C 180,E1 14582.807,E2 14582.807} C_VEL
LIN {X 0,Y 306.227,Z 617.636,A -85,B 0,C 180,E1 14578.316,E2 14578.316} C_VEL
LIN {X 0,Y 306.271,Z 617.904,A -85,B 0,C 180,E1 14574.003,E2 14574.003} C_VEL
LIN {X 0,Y 308.666,Z 622.99,A -85,B 0,C 180,E1 14569.737,E2 14569.737} C_VEL
LIN {X 0,Y 310.808,Z 627.681,A -85,B 0,C 180,E1 14566.607,E2 14566.607} C_VEL
LIN {X 0,Y 312.785,Z 632.147,A -85,B 0,C 180,E1 14564.043,E2 14564.043} C_VEL
LIN {X 0,Y 314.59,Z 636.444,A -85,B 0,C 180,E1 14561.852,E2 14561.852} C_VEL
LIN {X 0,Y 317.106,Z 642.275,A -85,B 0,C 180,E1 14559.127,E2 14559.127} C_VEL
LIN {X 0,Y 320.756,Z 652.366,A -85,B 0,C 180,E1 14555.108,E2 14555.108} C_VEL
LIN {X 0,Y 324.105,Z 662.732,A -85,B 0,C 180,E1 14551.548,E2 14551.548} C_VEL
LIN {X 0,Y 327.199,Z 674.2,A -85,B 0,C 180,E1 14548.085,E2 14548.085} C_VEL
LIN {X 0,Y 329.248,Z 683.731,A -85,B 0,C 180,E1 14545.492,E2 14545.492} C_VEL
LIN {X 0,Y 324.769,Z 705.69,A -85,B 0,C 180,E1 14541.442,E2 14541.442} C_VEL
LIN {X 0,Y 330.363,Z 734.564,A -85,B 0,C 180,E1 14539.707,E2 14539.707} C_VEL
LIN {X 0,Y 332.653,Z 749.838,A -85,B 0,C 180,E1 14538.939,E2 14538.939} C_VEL
LIN {X 0,Y 328.812,Z 839.526,A -85,B 0,C 180,E1 14536.79,E2 14536.79} C_VEL
LIN {X 0,Y 327.669,Z 855.807,A -85,B 0,C 180,E1 14536.075,E2 14536.075} C_VEL
LIN {X 0,Y 326.051,Z 870.875,A -85,B 0,C 180,E1 14535.103,E2 14535.103} C_VEL
LIN {X 0,Y 323.828,Z 885.979,A -85,B 0,C 180,E1 14533.759,E2 14533.759} C_VEL
LIN {X 0,Y 321.415,Z 899.233,A -85,B 0,C 180,E1 14532.216,E2 14532.216} C_VEL
LIN {X 0,Y 318.635,Z 912.168,A -85,B 0,C 180,E1 14530.272,E2 14530.272} C_VEL
LIN {X 0,Y 316.048,Z 922.885,A -85,B 0,C 180,E1 14528.206,E2 14528.206} C_VEL
LIN {X 0,Y 313.374,Z 932.933,A -85,B 0,C 180,E1 14525.724,E2 14525.724} C_VEL
LIN {X 0,Y 311.07,Z 940.901,A -85,B 0,C 180,E1 14523.122,E2 14523.122} C_VEL
LIN {X 0,Y 309.157,Z 947.3,A -85,B 0,C 180,E1 14520.3,E2 14520.3} C_VEL
LIN {X 0,Y 307.699,Z 951.908,A -85,B 0,C 180,E1 14517.269,E2 14517.269} C_VEL
LIN {X 0,Y 306.841,Z 954.441,A -85,B 0,C 180,E1 14514.446,E2 14514.446} C_VEL
LIN {X 0,Y 306.328,Z 955.335,A -85,B 0,C 180,E1 14511.242,E2 14511.242} C_VEL
LIN {X 0,Y 306.228,Z 954.405,A -85,B 0,C 180,E1 14508.267,E2 14508.267} C_VEL
LIN {X 0,Y 306.496,Z 951.514,A -85,B 0,C 180,E1 14505.128,E2 14505.128} C_VEL
LIN {X 0,Y 307.097,Z 947.226,A -85,B 0,C 180,E1 14502.377,E2 14502.377} C_VEL
LIN {X 0,Y 308.17,Z 940.762,A -85,B 0,C 180,E1 14499.482,E2 14499.482} C_VEL
LIN {X 0,Y 309.582,Z 932.795,A -85,B 0,C 180,E1 14496.863,E2 14496.863} C_VEL
LIN {X 0,Y 311.319,Z 923.198,A -85,B 0,C 180,E1 14494.42,E2 14494.42} C_VEL
LIN {X 0,Y 313.242,Z 911.931,A -85,B 0,C 180,E1 14492.195,E2 14492.195} C_VEL
LIN {X 0,Y 315.067,Z 900.275,A -85,B 0,C 180,E1 14490.363,E2 14490.363} C_VEL
LIN {X 0,Y 317.048,Z 886.117,A -85,B 0,C 180,E1 14488.634,E2 14488.634} C_VEL
LIN {X 0,Y 318.684,Z 871.874,A -85,B 0,C 180,E1 14487.302,E2 14487.302} C_VEL
LIN {X 0,Y 320.041,Z 856.515,A -85,B 0,C 180,E1 14486.238,E2 14486.238} C_VEL
LIN {X 0,Y 320.958,Z 840.55,A -85,B 0,C 180,E1 14485.488,E2 14485.488} C_VEL
LIN {X 0,Y 321.769,Z 815.175,A -85,B 0,C 180,E1 14484.81,E2 14484.81} C_VEL
LIN {X 0,Y 323.919,Z 744.866,A -85,B 0,C 180,E1 14483.191,E2 14483.191} C_VEL
LIN {X 0,Y 317.738,Z 705.466,A -85,B 0,C 180,E1 14481.54,E2 14481.54} C_VEL
LIN {X 0,Y 321.986,Z 678.51,A -85,B 0,C 180,E1 14476.715,E2 14476.715} C_VEL
LIN {X 0,Y 322.769,Z 672.719,A -85,B 0,C 180,E1 14475.651,E2 14475.651} C_VEL
LIN {X 0,Y 318.857,Z 656.91,A -85,B 0,C 180,E1 14471.914,E2 14471.914} C_VEL
LIN {X 0,Y 314.771,Z 642.702,A -85,B 0,C 180,E1 14468.28,E2 14468.28} C_VEL
LIN {X 0,Y 311.069,Z 631.353,A -85,B 0,C 180,E1 14465.126,E2 14465.126} C_VEL
LIN {X 0,Y 309.309,Z 629.173,A -85,B 0,C 180,E1 14464.316,E2 14464.316} C_VEL
LIN {X 0,Y 301.323,Z 625.489,A -85,B 0,C 180,E1 14461.983,E2 14461.983} C_VEL
LIN {X 0,Y 300.105,Z 623.936,A -85,B 0,C 180,E1 14461.371,E2 14461.371} C_VEL
LIN {X 0,Y 298.304,Z 618.722,A -85,B 0,C 180,E1 14459.593,E2 14459.593} C_VEL
LIN {X 0,Y 298.284,Z 618.644,A -85,B 0,C 180,E1 14455.026,E2 14455.026} C_VEL
LIN {X 0,Y 298.289,Z 618.639,A -85,B 0,C 180,E1 14450.44,E2 14450.44} C_VEL
LIN {X 0,Y 298.293,Z 618.618,A -85,B 0,C 180,E1 14445.796,E2 14445.796} C_VEL
LIN {X 0,Y 298.301,Z 618.603,A -85,B 0,C 180,E1 14441.324,E2 14441.324} C_VEL
LIN {X 0,Y 298.286,Z 618.64,A -85,B 0,C 180,E1 14436.761,E2 14436.761} C_VEL
LIN {X 0,Y 298.273,Z 618.614,A -85,B 0,C 180,E1 14432.208,E2 14432.208} C_VEL
LIN {X 0,Y 298.274,Z 618.613,A -85,B 0,C 180,E1 14427.751,E2 14427.751} C_VEL
LIN {X 0,Y 298.289,Z 618.63,A -85,B 0,C 180,E1 14423.091,E2 14423.091} C_VEL
LIN {X 0,Y 298.289,Z 618.595,A -85,B 0,C 180,E1 14418.569,E2 14418.569} C_VEL
LIN {X 0,Y 298.287,Z 618.64,A -85,B 0,C 180,E1 14413.966,E2 14413.966} C_VEL
LIN {X 0,Y 298.265,Z 618.593,A -85,B 0,C 180,E1 14409.455,E2 14409.455} C_VEL
LIN {X 0,Y 298.266,Z 618.641,A -85,B 0,C 180,E1 14404.808,E2 14404.808} C_VEL
LIN {X 0,Y 298.274,Z 618.594,A -85,B 0,C 180,E1 14400.192,E2 14400.192} C_VEL
LIN {X 0,Y 298.29,Z 618.636,A -85,B 0,C 180,E1 14395.579,E2 14395.579} C_VEL
LIN {X 0,Y 298.279,Z 618.612,A -85,B 0,C 180,E1 14391.13,E2 14391.13} C_VEL
LIN {X 0,Y 298.262,Z 618.615,A -85,B 0,C 180,E1 14386.626,E2 14386.626} C_VEL
LIN {X 0,Y 298.26,Z 618.647,A -85,B 0,C 180,E1 14382.037,E2 14382.037} C_VEL
LIN {X 0,Y 298.259,Z 618.631,A -85,B 0,C 180,E1 14377.533,E2 14377.533} C_VEL
LIN {X 0,Y 298.276,Z 618.619,A -85,B 0,C 180,E1 14373.085,E2 14373.085} C_VEL
LIN {X 0,Y 298.289,Z 618.62,A -85,B 0,C 180,E1 14368.698,E2 14368.698} C_VEL
LIN {X 0,Y 298.303,Z 618.894,A -85,B 0,C 180,E1 14365.961,E2 14365.961} C_VEL
LIN {X 0,Y 302.992,Z 630.431,A -85,B 0,C 180,E1 14362.614,E2 14362.614} C_VEL
LIN {X 0,Y 308.091,Z 643.446,A -85,B 0,C 180,E1 14359.284,E2 14359.284} C_VEL
LIN {X 0,Y 313.786,Z 659.511,A -85,B 0,C 180,E1 14355.62,E2 14355.62} C_VEL
LIN {X 0,Y 319.395,Z 676.984,A -85,B 0,C 180,E1 14352.062,E2 14352.062} C_VEL
LIN {X 0,Y 321.36,Z 684.443,A -85,B 0,C 180,E1 14350.68,E2 14350.68} C_VEL
LIN {X 0,Y 319.268,Z 696.12,A -85,B 0,C 180,E1 14349.192,E2 14349.192} C_VEL
LIN {X 0,Y 322.142,Z 731.016,A -85,B 0,C 180,E1 14348.012,E2 14348.012} C_VEL
LIN {X 0,Y 317.336,Z 884.441,A -85,B 0,C 180,E1 14344.669,E2 14344.669} C_VEL
LIN {X 0,Y 315.967,Z 902.674,A -85,B 0,C 180,E1 14343.97,E2 14343.97} C_VEL
LIN {X 0,Y 313.935,Z 920.782,A -85,B 0,C 180,E1 14342.945,E2 14342.945} C_VEL
LIN {X 0,Y 311.544,Z 938.039,A -85,B 0,C 180,E1 14341.612,E2 14341.612} C_VEL
LIN {X 0,Y 309.003,Z 954.195,A -85,B 0,C 180,E1 14339.996,E2 14339.996} C_VEL
LIN {X 0,Y 306.302,Z 969.752,A -85,B 0,C 180,E1 14338.039,E2 14338.039} C_VEL
LIN {X 0,Y 303.674,Z 984.261,A -85,B 0,C 180,E1 14335.761,E2 14335.761} C_VEL
LIN {X 0,Y 301.353,Z 997.466,A -85,B 0,C 180,E1 14333.212,E2 14333.212} C_VEL
LIN {X 0,Y 299.387,Z 1009.632,A -85,B 0,C 180,E1 14330.324,E2 14330.324} C_VEL
LIN {X 0,Y 298.028,Z 1019.727,A -85,B 0,C 180,E1 14327.373,E2 14327.373} C_VEL
LIN {X 0,Y 297.254,Z 1028.409,A -85,B 0,C 180,E1 14324.215,E2 14324.215} C_VEL
LIN {X 0,Y 297.029,Z 1035.58,A -85,B 0,C 180,E1 14320.866,E2 14320.866} C_VEL
LIN {X 0,Y 297.277,Z 1040.832,A -85,B 0,C 180,E1 14317.538,E2 14317.538} C_VEL
LIN {X 0,Y 297.678,Z 1044.095,A -85,B 0,C 180,E1 14314.431,E2 14314.431} C_VEL
LIN {X 0,Y 297.965,Z 1045.806,A -85,B 0,C 180,E1 14311.346,E2 14311.346} C_VEL
LIN {X 0,Y 297.913,Z 1046.022,A -85,B 0,C 180,E1 14308.462,E2 14308.462} C_VEL
LIN {X 0,Y 297.538,Z 1044.8,A -85,B 0,C 180,E1 14305.374,E2 14305.374} C_VEL
LIN {X 0,Y 297.069,Z 1041.879,A -85,B 0,C 180,E1 14302.068,E2 14302.068} C_VEL
LIN {X 0,Y 296.845,Z 1037.286,A -85,B 0,C 180,E1 14298.735,E2 14298.735} C_VEL
LIN {X 0,Y 297.17,Z 1030.953,A -85,B 0,C 180,E1 14295.384,E2 14295.384} C_VEL
LIN {X 0,Y 298.185,Z 1022.741,A -85,B 0,C 180,E1 14292.032,E2 14292.032} C_VEL
LIN {X 0,Y 300.056,Z 1012.415,A -85,B 0,C 180,E1 14288.703,E2 14288.703} C_VEL
LIN {X 0,Y 302.457,Z 1001.244,A -85,B 0,C 180,E1 14285.801,E2 14285.801} C_VEL
LIN {X 0,Y 305.368,Z 988.699,A -85,B 0,C 180,E1 14283.138,E2 14283.138} C_VEL
LIN {X 0,Y 308.711,Z 974.668,A -85,B 0,C 180,E1 14280.721,E2 14280.721} C_VEL
LIN {X 0,Y 312.171,Z 959.556,A -85,B 0,C 180,E1 14278.636,E2 14278.636} C_VEL
LIN {X 0,Y 315.545,Z 943.419,A -85,B 0,C 180,E1 14276.866,E2 14276.866} C_VEL
LIN {X 0,Y 318.731,Z 926.195,A -85,B 0,C 180,E1 14275.403,E2 14275.403} C_VEL
LIN {X 0,Y 321.398,Z 909.048,A -85,B 0,C 180,E1 14274.317,E2 14274.317} C_VEL
LIN {X 0,Y 323.473,Z 891.033,A -85,B 0,C 180,E1 14273.507,E2 14273.507} C_VEL
LIN {X 0,Y 324.65,Z 872.376,A -85,B 0,C 180,E1 14272.969,E2 14272.969} C_VEL
LIN {X 0,Y 330.121,Z 729.488,A -85,B 0,C 180,E1 14269.814,E2 14269.814} C_VEL
LIN {X 0,Y 327.344,Z 699.935,A -85,B 0,C 180,E1 14268.537,E2 14268.537} C_VEL
LIN {X 0,Y 327.159,Z 695.944,A -85,B 0,C 180,E1 14268.281,E2 14268.281} C_VEL
LIN {X 0,Y 328.032,Z 691.564,A -85,B 0,C 180,E1 14267.653,E2 14267.653} C_VEL
LIN {X 0,Y 324.212,Z 678.533,A -85,B 0,C 180,E1 14264.57,E2 14264.57} C_VEL
LIN {X 0,Y 319.995,Z 666.441,A -85,B 0,C 180,E1 14261.246,E2 14261.246} C_VEL
LIN {X 0,Y 315.864,Z 655.989,A -85,B 0,C 180,E1 14257.886,E2 14257.886} C_VEL
LIN {X 0,Y 312.259,Z 647.713,A -85,B 0,C 180,E1 14254.747,E2 14254.747} C_VEL
LIN {X 0,Y 309.238,Z 641.038,A -85,B 0,C 180,E1 14251.804,E2 14251.804} C_VEL
LIN {X 0,Y 307.418,Z 637.089,A -85,B 0,C 180,E1 14249.843,E2 14249.843} C_VEL
LIN {X 0,Y 305.24,Z 632.584,A -85,B 0,C 180,E1 14247.296,E2 14247.296} C_VEL
LIN {X 0,Y 303.058,Z 628.186,A -85,B 0,C 180,E1 14244.356,E2 14244.356} C_VEL
LIN {X 0,Y 300.582,Z 623.392,A -85,B 0,C 180,E1 14240.239,E2 14240.239} C_VEL
LIN {X 0,Y 298.277,Z 618.791,A -85,B 0,C 180,E1 14233.793,E2 14233.793} C_VEL
LIN {X 0,Y 298.263,Z 618.614,A -85,B 0,C 180,E1 14229.259,E2 14229.259} C_VEL
LIN {X 0,Y 298.272,Z 618.613,A -85,B 0,C 180,E1 14224.807,E2 14224.807} C_VEL
LIN {X 0,Y 298.335,Z 618.981,A -85,B 0,C 180,E1 14220.576,E2 14220.576} C_VEL
LIN {X 0,Y 300.845,Z 624,A -85,B 0,C 180,E1 14213.895,E2 14213.895} C_VEL
LIN {X 0,Y 303.051,Z 628.603,A -85,B 0,C 180,E1 14209.929,E2 14209.929} C_VEL
LIN {X 0,Y 305.15,Z 633.376,A -85,B 0,C 180,E1 14206.694,E2 14206.694} C_VEL
LIN {X 0,Y 307.053,Z 637.782,A -85,B 0,C 180,E1 14204.125,E2 14204.125} C_VEL
LIN {X 0,Y 308.799,Z 642.063,A -85,B 0,C 180,E1 14201.89,E2 14201.89} C_VEL
LIN {X 0,Y 311.21,Z 647.922,A -85,B 0,C 180,E1 14199.107,E2 14199.107} C_VEL
LIN {X 0,Y 314.486,Z 657.092,A -85,B 0,C 180,E1 14195.386,E2 14195.386} C_VEL
LIN {X 0,Y 317.658,Z 667.251,A -85,B 0,C 180,E1 14191.803,E2 14191.803} C_VEL
LIN {X 0,Y 320.557,Z 678.339,A -85,B 0,C 180,E1 14188.378,E2 14188.378} C_VEL
LIN {X 0,Y 322.302,Z 687.198,A -85,B 0,C 180,E1 14185.924,E2 14185.924} C_VEL
LIN {X 0,Y 318.349,Z 705.178,A -85,B 0,C 180,E1 14182.53,E2 14182.53} C_VEL
LIN {X 0,Y 323.319,Z 730.97,A -85,B 0,C 180,E1 14180.871,E2 14180.871} C_VEL
LIN {X 0,Y 326.443,Z 750.895,A -85,B 0,C 180,E1 14179.804,E2 14179.804} C_VEL
LIN {X 0,Y 322.423,Z 840.091,A -85,B 0,C 180,E1 14177.632,E2 14177.632} C_VEL
LIN {X 0,Y 321.228,Z 856.307,A -85,B 0,C 180,E1 14176.911,E2 14176.911} C_VEL
LIN {X 0,Y 319.497,Z 871.648,A -85,B 0,C 180,E1 14175.907,E2 14175.907} C_VEL
LIN {X 0,Y 317.203,Z 886.462,A -85,B 0,C 180,E1 14174.571,E2 14174.571} C_VEL
LIN {X 0,Y 314.633,Z 899.94,A -85,B 0,C 180,E1 14172.985,E2 14172.985} C_VEL
LIN {X 0,Y 311.684,Z 912.978,A -85,B 0,C 180,E1 14170.997,E2 14170.997} C_VEL
LIN {X 0,Y 308.943,Z 923.751,A -85,B 0,C 180,E1 14168.892,E2 14168.892} C_VEL
LIN {X 0,Y 306.202,Z 933.47,A -85,B 0,C 180,E1 14166.462,E2 14166.462} C_VEL
LIN {X 0,Y 303.88,Z 941.127,A -85,B 0,C 180,E1 14163.987,E2 14163.987} C_VEL
LIN {X 0,Y 301.761,Z 947.708,A -85,B 0,C 180,E1 14161.124,E2 14161.124} C_VEL
LIN {X 0,Y 300.207,Z 952.366,A -85,B 0,C 180,E1 14158.225,E2 14158.225} C_VEL
LIN {X 0,Y 299.088,Z 955.419,A -85,B 0,C 180,E1 14155.046,E2 14155.046} C_VEL
LIN {X 0,Y 298.504,Z 956.53,A -85,B 0,C 180,E1 14152.033,E2 14152.033} C_VEL
LIN {X 0,Y 298.305,Z 955.853,A -85,B 0,C 180,E1 14148.77,E2 14148.77} C_VEL
LIN {X 0,Y 298.492,Z 953.443,A -85,B 0,C 180,E1 14145.743,E2 14145.743} C_VEL
LIN {X 0,Y 299.072,Z 949.279,A -85,B 0,C 180,E1 14142.747,E2 14142.747} C_VEL
LIN {X 0,Y 300.018,Z 943.642,A -85,B 0,C 180,E1 14139.979,E2 14139.979} C_VEL
LIN {X 0,Y 301.403,Z 936.112,A -85,B 0,C 180,E1 14137.242,E2 14137.242} C_VEL
LIN {X 0,Y 303.105,Z 927.071,A -85,B 0,C 180,E1 14134.73,E2 14134.73} C_VEL
LIN {X 0,Y 305.024,Z 916.582,A -85,B 0,C 180,E1 14132.442,E2 14132.442} C_VEL
LIN {X 0,Y 306.969,Z 904.939,A -85,B 0,C 180,E1 14130.437,E2 14130.437} C_VEL
LIN {X 0,Y 309.053,Z 891.284,A -85,B 0,C 180,E1 14128.591,E2 14128.591} C_VEL
LIN {X 0,Y 310.835,Z 877.299,A -85,B 0,C 180,E1 14127.142,E2 14127.142} C_VEL
LIN {X 0,Y 312.363,Z 862.27,A -85,B 0,C 180,E1 14125.961,E2 14125.961} C_VEL
LIN {X 0,Y 313.527,Z 845.446,A -85,B 0,C 180,E1 14125.049,E2 14125.049} C_VEL
LIN {X 0,Y 314.157,Z 828.55,A -85,B 0,C 180,E1 14124.495,E2 14124.495} C_VEL
LIN {X 0,Y 316.797,Z 745.878,A -85,B 0,C 180,E1 14122.545,E2 14122.545} C_VEL
LIN {X 0,Y 310.521,Z 705.638,A -85,B 0,C 180,E1 14120.828,E2 14120.828} C_VEL
LIN {X 0,Y 314.859,Z 679.247,A -85,B 0,C 180,E1 14116.034,E2 14116.034} C_VEL
LIN {X 0,Y 315.356,Z 675.115,A -85,B 0,C 180,E1 14115.248,E2 14115.248} C_VEL
LIN {X 0,Y 311.517,Z 659.513,A -85,B 0,C 180,E1 14111.472,E2 14111.472} C_VEL
LIN {X 0,Y 307.458,Z 645.315,A -85,B 0,C 180,E1 14107.736,E2 14107.736} C_VEL
LIN {X 0,Y 303.352,Z 632.791,A -85,B 0,C 180,E1 14104.135,E2 14104.135} C_VEL
LIN {X 0,Y 300.105,Z 623.936,A -85,B 0,C 180,E1 14101.371,E2 14101.371} C_VEL
LIN {X 0,Y 298.381,Z 621.8,A -85,B 0,C 180,E1 14100.497,E2 14100.497} C_VEL
LIN {X 0,Y 294.454,Z 620.157,A -85,B 0,C 180,E1 14099.258,E2 14099.258} C_VEL
LIN {X 0,Y 290.966,Z 619.605,A -85,B 0,C 180,E1 14097.931,E2 14097.931} C_VEL
LIN {X 0,Y 290.337,Z 619.565,A -85,B 0,C 180,E1 14097.2,E2 14097.2} C_VEL
LIN {X 0,Y 290.343,Z 619.607,A -85,B 0,C 180,E1 14092.692,E2 14092.692} C_VEL
LIN {X 0,Y 290.354,Z 619.605,A -85,B 0,C 180,E1 14088.058,E2 14088.058} C_VEL
LIN {X 0,Y 290.356,Z 619.627,A -85,B 0,C 180,E1 14083.398,E2 14083.398} C_VEL
LIN {X 0,Y 290.348,Z 619.613,A -85,B 0,C 180,E1 14078.811,E2 14078.811} C_VEL
LIN {X 0,Y 290.334,Z 619.589,A -85,B 0,C 180,E1 14074.149,E2 14074.149} C_VEL
LIN {X 0,Y 290.348,Z 619.63,A -85,B 0,C 180,E1 14069.502,E2 14069.502} C_VEL
LIN {X 0,Y 290.351,Z 619.586,A -85,B 0,C 180,E1 14064.843,E2 14064.843} C_VEL
LIN {X 0,Y 290.352,Z 619.617,A -85,B 0,C 180,E1 14060.354,E2 14060.354} C_VEL
LIN {X 0,Y 290.332,Z 619.595,A -85,B 0,C 180,E1 14055.788,E2 14055.788} C_VEL
LIN {X 0,Y 290.326,Z 619.606,A -85,B 0,C 180,E1 14051.12,E2 14051.12} C_VEL
LIN {X 0,Y 290.336,Z 619.608,A -85,B 0,C 180,E1 14046.526,E2 14046.526} C_VEL
LIN {X 0,Y 290.348,Z 619.59,A -85,B 0,C 180,E1 14041.974,E2 14041.974} C_VEL
LIN {X 0,Y 290.344,Z 619.624,A -85,B 0,C 180,E1 14037.435,E2 14037.435} C_VEL
LIN {X 0,Y 290.323,Z 619.588,A -85,B 0,C 180,E1 14032.878,E2 14032.878} C_VEL
LIN {X 0,Y 290.321,Z 619.63,A -85,B 0,C 180,E1 14028.277,E2 14028.277} C_VEL
LIN {X 0,Y 290.322,Z 619.614,A -85,B 0,C 180,E1 14023.802,E2 14023.802} C_VEL
LIN {X 0,Y 290.343,Z 619.599,A -85,B 0,C 180,E1 14019.225,E2 14019.225} C_VEL
LIN {X 0,Y 290.346,Z 619.608,A -85,B 0,C 180,E1 14014.722,E2 14014.722} C_VEL
LIN {X 0,Y 290.334,Z 619.617,A -85,B 0,C 180,E1 14010.21,E2 14010.21} C_VEL
LIN {X 0,Y 290.356,Z 619.908,A -85,B 0,C 180,E1 14007.42,E2 14007.42} C_VEL
LIN {X 0,Y 295.127,Z 631.452,A -85,B 0,C 180,E1 14003.879,E2 14003.879} C_VEL
LIN {X 0,Y 300.415,Z 644.808,A -85,B 0,C 180,E1 14000.281,E2 14000.281} C_VEL
LIN {X 0,Y 306.081,Z 660.757,A -85,B 0,C 180,E1 13996.486,E2 13996.486} C_VEL
LIN {X 0,Y 311.536,Z 677.835,A -85,B 0,C 180,E1 13992.876,E2 13992.876} C_VEL
LIN {X 0,Y 314.029,Z 686.583,A -85,B 0,C 180,E1 13991.17,E2 13991.17} C_VEL
LIN {X 0,Y 312.236,Z 696.247,A -85,B 0,C 180,E1 13989.916,E2 13989.916} C_VEL
LIN {X 0,Y 315.086,Z 731.758,A -85,B 0,C 180,E1 13988.684,E2 13988.684} C_VEL
LIN {X 0,Y 310.102,Z 883.947,A -85,B 0,C 180,E1 13985.299,E2 13985.299} C_VEL
LIN {X 0,Y 308.684,Z 902.247,A -85,B 0,C 180,E1 13984.58,E2 13984.58} C_VEL
LIN {X 0,Y 306.538,Z 920.707,A -85,B 0,C 180,E1 13983.509,E2 13983.509} C_VEL
LIN {X 0,Y 304.127,Z 937.465,A -85,B 0,C 180,E1 13982.182,E2 13982.182} C_VEL
LIN {X 0,Y 301.448,Z 953.904,A -85,B 0,C 180,E1 13980.497,E2 13980.497} C_VEL
LIN {X 0,Y 298.656,Z 969.346,A -85,B 0,C 180,E1 13978.495,E2 13978.495} C_VEL
LIN {X 0,Y 295.935,Z 983.756,A -85,B 0,C 180,E1 13976.163,E2 13976.163} C_VEL
LIN {X 0,Y 293.484,Z 997.131,A -85,B 0,C 180,E1 13973.491,E2 13973.491} C_VEL
LIN {X 0,Y 291.434,Z 1009.335,A -85,B 0,C 180,E1 13970.484,E2 13970.484} C_VEL
LIN {X 0,Y 290.05,Z 1019.289,A -85,B 0,C 180,E1 13967.452,E2 13967.452} C_VEL
LIN {X 0,Y 289.275,Z 1027.837,A -85,B 0,C 180,E1 13964.206,E2 13964.206} C_VEL
LIN {X 0,Y 289.074,Z 1034.871,A -85,B 0,C 180,E1 13960.765,E2 13960.765} C_VEL
LIN {X 0,Y 289.364,Z 1039.975,A -85,B 0,C 180,E1 13957.346,E2 13957.346} C_VEL
LIN {X 0,Y 289.789,Z 1043.132,A -85,B 0,C 180,E1 13954.155,E2 13954.155} C_VEL
LIN {X 0,Y 290.069,Z 1044.7,A -85,B 0,C 180,E1 13950.988,E2 13950.988} C_VEL
LIN {X 0,Y 289.958,Z 1044.757,A -85,B 0,C 180,E1 13948.024,E2 13948.024} C_VEL
LIN {X 0,Y 289.523,Z 1043.368,A -85,B 0,C 180,E1 13944.849,E2 13944.849} C_VEL
LIN {X 0,Y 289.039,Z 1040.274,A -85,B 0,C 180,E1 13941.446,E2 13941.446} C_VEL
LIN {X 0,Y 288.889,Z 1035.166,A -85,B 0,C 180,E1 13937.812,E2 13937.812} C_VEL
LIN {X 0,Y 289.442,Z 1028.103,A -85,B 0,C 180,E1 13934.163,E2 13934.163} C_VEL
LIN {X 0,Y 290.77,Z 1019.474,A -85,B 0,C 180,E1 13930.725,E2 13930.725} C_VEL
LIN {X 0,Y 292.858,Z 1009.394,A -85,B 0,C 180,E1 13927.519,E2 13927.519} C_VEL
LIN {X 0,Y 295.587,Z 997.833,A -85,B 0,C 180,E1 13924.558,E2 13924.558} C_VEL
LIN {X 0,Y 298.83,Z 984.758,A -85,B 0,C 180,E1 13921.851,E2 13921.851} C_VEL
LIN {X 0,Y 302.357,Z 970.688,A -85,B 0,C 180,E1 13919.496,E2 13919.496} C_VEL
LIN {X 0,Y 306.088,Z 954.95,A -85,B 0,C 180,E1 13917.386,E2 13917.386} C_VEL
LIN {X 0,Y 309.536,Z 938.918,A -85,B 0,C 180,E1 13915.69,E2 13915.69} C_VEL
LIN {X 0,Y 312.671,Z 922.341,A -85,B 0,C 180,E1 13914.336,E2 13914.336} C_VEL
LIN {X 0,Y 315.407,Z 904.612,A -85,B 0,C 180,E1 13913.263,E2 13913.263} C_VEL
LIN {X 0,Y 317.387,Z 886.427,A -85,B 0,C 180,E1 13912.505,E2 13912.505} C_VEL
LIN {X 0,Y 318.55,Z 864.449,A -85,B 0,C 180,E1 13911.936,E2 13911.936} C_VEL
LIN {X 0,Y 323.974,Z 730.21,A -85,B 0,C 180,E1 13908.914,E2 13908.914} C_VEL
LIN {X 0,Y 321.332,Z 701.227,A -85,B 0,C 180,E1 13907.622,E2 13907.622} C_VEL
LIN {X 0,Y 320.967,Z 696.469,A -85,B 0,C 180,E1 13907.348,E2 13907.348} C_VEL
LIN {X 0,Y 321.306,Z 695.063,A -85,B 0,C 180,E1 13907.161,E2 13907.161} C_VEL
LIN {X 0,Y 317.678,Z 682.422,A -85,B 0,C 180,E1 13904.073,E2 13904.073} C_VEL
LIN {X 0,Y 313.709,Z 670.878,A -85,B 0,C 180,E1 13900.797,E2 13900.797} C_VEL
LIN {X 0,Y 309.771,Z 660.731,A -85,B 0,C 180,E1 13897.437,E2 13897.437} C_VEL
LIN {X 0,Y 305.858,Z 651.316,A -85,B 0,C 180,E1 13893.761,E2 13893.761} C_VEL
LIN {X 0,Y 303.23,Z 645.864,A -85,B 0,C 180,E1 13891.177,E2 13891.177} C_VEL
LIN {X 0,Y 301.841,Z 642.7,A -85,B 0,C 180,E1 13889.575,E2 13889.575} C_VEL
LIN {X 0,Y 299.711,Z 638.25,A -85,B 0,C 180,E1 13886.981,E2 13886.981} C_VEL
LIN {X 0,Y 297.756,Z 634.134,A -85,B 0,C 180,E1 13884.184,E2 13884.184} C_VEL
LIN {X 0,Y 295.422,Z 629.501,A -85,B 0,C 180,E1 13880.195,E2 13880.195} C_VEL
LIN {X 0,Y 292.98,Z 624.764,A -85,B 0,C 180,E1 13873.619,E2 13873.619} C_VEL
LIN {X 0,Y 292.044,Z 623.619,A -85,B 0,C 180,E1 13868.465,E2 13868.465} C_VEL
LIN {X 0,Y 292.417,Z 624.109,A -85,B 0,C 180,E1 13863.209,E2 13863.209} C_VEL
LIN {X 0,Y 293.112,Z 625.251,A -85,B 0,C 180,E1 13860.195,E2 13860.195} C_VEL
LIN {X 0,Y 295.414,Z 629.897,A -85,B 0,C 180,E1 13853.977,E2 13853.977} C_VEL
LIN {X 0,Y 297.548,Z 634.574,A -85,B 0,C 180,E1 13849.924,E2 13849.924} C_VEL
LIN {X 0,Y 299.465,Z 638.927,A -85,B 0,C 180,E1 13846.877,E2 13846.877} C_VEL
LIN {X 0,Y 301.298,Z 643.382,A -85,B 0,C 180,E1 13844.209,E2 13844.209} C_VEL
LIN {X 0,Y 303.868,Z 649.477,A -85,B 0,C 180,E1 13840.988,E2 13840.988} C_VEL
LIN {X 0,Y 307.093,Z 658.461,A -85,B 0,C 180,E1 13837.001,E2 13837.001} C_VEL
LIN {X 0,Y 310.306,Z 668.563,A -85,B 0,C 180,E1 13833.194,E2 13833.194} C_VEL
LIN {X 0,Y 313.133,Z 679.147,A -85,B 0,C 180,E1 13829.701,E2 13829.701} C_VEL
LIN {X 0,Y 315.478,Z 690.266,A -85,B 0,C 180,E1 13826.464,E2 13826.464} C_VEL
LIN {X 0,Y 312.044,Z 705.405,A -85,B 0,C 180,E1 13823.581,E2 13823.581} C_VEL
LIN {X 0,Y 317.582,Z 734.315,A -85,B 0,C 180,E1 13821.681,E2 13821.681} C_VEL
LIN {X 0,Y 320.295,Z 752.293,A -85,B 0,C 180,E1 13820.695,E2 13820.695} C_VEL
LIN {X 0,Y 316.117,Z 840.82,A -85,B 0,C 180,E1 13818.506,E2 13818.506} C_VEL
LIN {X 0,Y 314.85,Z 857.147,A -85,B 0,C 180,E1 13817.768,E2 13817.768} C_VEL
LIN {X 0,Y 313.02,Z 872.551,A -85,B 0,C 180,E1 13816.743,E2 13816.743} C_VEL
LIN {X 0,Y 310.564,Z 887.622,A -85,B 0,C 180,E1 13815.358,E2 13815.358} C_VEL
LIN {X 0,Y 307.892,Z 900.901,A -85,B 0,C 180,E1 13813.765,E2 13813.765} C_VEL
LIN {X 0,Y 304.795,Z 913.852,A -85,B 0,C 180,E1 13811.753,E2 13811.753} C_VEL
LIN {X 0,Y 301.908,Z 924.588,A -85,B 0,C 180,E1 13809.622,E2 13809.622} C_VEL
LIN {X 0,Y 298.866,Z 934.739,A -85,B 0,C 180,E1 13807.027,E2 13807.027} C_VEL
LIN {X 0,Y 296.425,Z 942.303,A -85,B 0,C 180,E1 13804.518,E2 13804.518} C_VEL
LIN {X 0,Y 294.149,Z 948.922,A -85,B 0,C 180,E1 13801.565,E2 13801.565} C_VEL
LIN {X 0,Y 292.48,Z 953.571,A -85,B 0,C 180,E1 13798.594,E2 13798.594} C_VEL
LIN {X 0,Y 291.285,Z 956.567,A -85,B 0,C 180,E1 13795.408,E2 13795.408} C_VEL
LIN {X 0,Y 290.623,Z 957.741,A -85,B 0,C 180,E1 13792.237,E2 13792.237} C_VEL
LIN {X 0,Y 290.389,Z 957.07,A -85,B 0,C 180,E1 13788.884,E2 13788.884} C_VEL
LIN {X 0,Y 290.568,Z 954.686,A -85,B 0,C 180,E1 13785.774,E2 13785.774} C_VEL
LIN {X 0,Y 291.159,Z 950.543,A -85,B 0,C 180,E1 13782.696,E2 13782.696} C_VEL
LIN {X 0,Y 292.18,Z 944.705,A -85,B 0,C 180,E1 13779.747,E2 13779.747} C_VEL
LIN {X 0,Y 293.688,Z 936.87,A -85,B 0,C 180,E1 13776.843,E2 13776.843} C_VEL
LIN {X 0,Y 295.479,Z 927.723,A -85,B 0,C 180,E1 13774.269,E2 13774.269} C_VEL
LIN {X 0,Y 297.588,Z 916.66,A -85,B 0,C 180,E1 13771.829,E2 13771.829} C_VEL
LIN {X 0,Y 299.707,Z 904.339,A -85,B 0,C 180,E1 13769.713,E2 13769.713} C_VEL
LIN {X 0,Y 301.693,Z 891.761,A -85,B 0,C 180,E1 13768.005,E2 13768.005} C_VEL
LIN {X 0,Y 303.563,Z 877.57,A -85,B 0,C 180,E1 13766.516,E2 13766.516} C_VEL
LIN {X 0,Y 305.106,Z 862.902,A -85,B 0,C 180,E1 13765.347,E2 13765.347} C_VEL
LIN {X 0,Y 306.322,Z 846.047,A -85,B 0,C 180,E1 13764.415,E2 13764.415} C_VEL
LIN {X 0,Y 306.983,Z 829.028,A -85,B 0,C 180,E1 13763.847,E2 13763.847} C_VEL
LIN {X 0,Y 309.714,Z 746.866,A -85,B 0,C 180,E1 13761.868,E2 13761.868} C_VEL
LIN {X 0,Y 303.365,Z 705.508,A -85,B 0,C 180,E1 13760.045,E2 13760.045} C_VEL
LIN {X 0,Y 307.945,Z 678.967,A -85,B 0,C 180,E1 13755.137,E2 13755.137} C_VEL
LIN {X 0,Y 307.675,Z 676.317,A -85,B 0,C 180,E1 13754.545,E2 13754.545} C_VEL
LIN {X 0,Y 303.942,Z 661.155,A -85,B 0,C 180,E1 13750.758,E2 13750.758} C_VEL
LIN {X 0,Y 300.036,Z 647.505,A -85,B 0,C 180,E1 13747.051,E2 13747.051} C_VEL
LIN {X 0,Y 296.135,Z 635.454,A -85,B 0,C 180,E1 13743.476,E2 13743.476} C_VEL
LIN {X 0,Y 291.567,Z 622.977,A -85,B 0,C 180,E1 13739.401,E2 13739.401} C_VEL
LIN {X 0,Y 290.372,Z 619.716,A -85,B 0,C 180,E1 13738.149,E2 13738.149} C_VEL
LIN {X 0,Y 290.337,Z 619.565,A -85,B 0,C 180,E1 13737.2,E2 13737.2} C_VEL
LIN {X 0,Y 289.467,Z 619.718,A -85,B 0,C 180,E1 13735.787,E2 13735.787} C_VEL
LIN {X 0,Y 285.609,Z 620.207,A -85,B 0,C 180,E1 13733.34,E2 13733.34} C_VEL
LIN {X 0,Y 282.658,Z 620.577,A -85,B 0,C 180,E1 13731.032,E2 13731.032} C_VEL
LIN {X 0,Y 282.419,Z 620.618,A -85,B 0,C 180,E1 13730.237,E2 13730.237} C_VEL
LIN {X 0,Y 282.415,Z 620.598,A -85,B 0,C 180,E1 13725.492,E2 13725.492} C_VEL
LIN {X 0,Y 282.402,Z 620.58,A -85,B 0,C 180,E1 13720.739,E2 13720.739} C_VEL
LIN {X 0,Y 282.401,Z 620.602,A -85,B 0,C 180,E1 13715.997,E2 13715.997} C_VEL
LIN {X 0,Y 282.415,Z 620.604,A -85,B 0,C 180,E1 13711.362,E2 13711.362} C_VEL
LIN {X 0,Y 282.414,Z 620.571,A -85,B 0,C 180,E1 13706.721,E2 13706.721} C_VEL
LIN {X 0,Y 282.399,Z 620.62,A -85,B 0,C 180,E1 13701.929,E2 13701.929} C_VEL
LIN {X 0,Y 282.393,Z 620.567,A -85,B 0,C 180,E1 13697.061,E2 13697.061} C_VEL
LIN {X 0,Y 282.412,Z 620.614,A -85,B 0,C 180,E1 13692.473,E2 13692.473} C_VEL
LIN {X 0,Y 282.404,Z 620.571,A -85,B 0,C 180,E1 13687.732,E2 13687.732} C_VEL
LIN {X 0,Y 282.387,Z 620.6,A -85,B 0,C 180,E1 13683.045,E2 13683.045} C_VEL
LIN {X 0,Y 282.385,Z 620.596,A -85,B 0,C 180,E1 13678.377,E2 13678.377} C_VEL
LIN {X 0,Y 282.41,Z 620.578,A -85,B 0,C 180,E1 13673.699,E2 13673.699} C_VEL
LIN {X 0,Y 282.4,Z 620.621,A -85,B 0,C 180,E1 13668.978,E2 13668.978} C_VEL
LIN {X 0,Y 282.381,Z 620.592,A -85,B 0,C 180,E1 13664.39,E2 13664.39} C_VEL
LIN {X 0,Y 282.382,Z 620.591,A -85,B 0,C 180,E1 13659.697,E2 13659.697} C_VEL
LIN {X 0,Y 282.398,Z 620.601,A -85,B 0,C 180,E1 13655.082,E2 13655.082} C_VEL
LIN {X 0,Y 282.418,Z 620.606,A -85,B 0,C 180,E1 13650.521,E2 13650.521} C_VEL
LIN {X 0,Y 282.446,Z 620.967,A -85,B 0,C 180,E1 13648.982,E2 13648.982} C_VEL
LIN {X 0,Y 287.359,Z 632.574,A -85,B 0,C 180,E1 13645.202,E2 13645.202} C_VEL
LIN {X 0,Y 292.465,Z 645.486,A -85,B 0,C 180,E1 13641.523,E2 13641.523} C_VEL
LIN {X 0,Y 297.921,Z 660.697,A -85,B 0,C 180,E1 13637.709,E2 13637.709} C_VEL
LIN {X 0,Y 303.263,Z 677.087,A -85,B 0,C 180,E1 13634.049,E2 13634.049} C_VEL
LIN {X 0,Y 306.699,Z 688.71,A -85,B 0,C 180,E1 13631.687,E2 13631.687} C_VEL
LIN {X 0,Y 305.254,Z 696.411,A -85,B 0,C 180,E1 13630.671,E2 13630.671} C_VEL
LIN {X 0,Y 308.074,Z 732.611,A -85,B 0,C 180,E1 13629.384,E2 13629.384} C_VEL
LIN {X 0,Y 302.924,Z 883.18,A -85,B 0,C 180,E1 13625.968,E2 13625.968} C_VEL
LIN {X 0,Y 301.463,Z 901.537,A -85,B 0,C 180,E1 13625.233,E2 13625.233} C_VEL
LIN {X 0,Y 299.262,Z 919.901,A -85,B 0,C 180,E1 13624.147,E2 13624.147} C_VEL
LIN {X 0,Y 296.684,Z 937.18,A -85,B 0,C 180,E1 13622.746,E2 13622.746} C_VEL
LIN {X 0,Y 293.901,Z 953.582,A -85,B 0,C 180,E1 13621.014,E2 13621.014} C_VEL
LIN {X 0,Y 290.901,Z 969.459,A -85,B 0,C 180,E1 13618.876,E2 13618.876} C_VEL
LIN {X 0,Y 288.212,Z 983.181,A -85,B 0,C 180,E1 13616.585,E2 13616.585} C_VEL
LIN {X 0,Y 285.754,Z 996.063,A -85,B 0,C 180,E1 13613.947,E2 13613.947} C_VEL
LIN {X 0,Y 283.628,Z 1008.137,A -85,B 0,C 180,E1 13610.903,E2 13610.903} C_VEL
LIN {X 0,Y 282.148,Z 1018.237,A -85,B 0,C 180,E1 13607.744,E2 13607.744} C_VEL
LIN {X 0,Y 281.328,Z 1026.772,A -85,B 0,C 180,E1 13604.406,E2 13604.406} C_VEL
LIN {X 0,Y 281.116,Z 1033.781,A -85,B 0,C 180,E1 13600.866,E2 13600.866} C_VEL
LIN {X 0,Y 281.428,Z 1038.859,A -85,B 0,C 180,E1 13597.349,E2 13597.349} C_VEL
LIN {X 0,Y 281.882,Z 1041.994,A -85,B 0,C 180,E1 13594.068,E2 13594.068} C_VEL
LIN {X 0,Y 282.163,Z 1043.46,A -85,B 0,C 180,E1 13591.016,E2 13591.016} C_VEL
LIN {X 0,Y 282.037,Z 1043.564,A -85,B 0,C 180,E1 13587.969,E2 13587.969} C_VEL
LIN {X 0,Y 281.563,Z 1042.208,A -85,B 0,C 180,E1 13584.703,E2 13584.703} C_VEL
LIN {X 0,Y 281.049,Z 1039.139,A -85,B 0,C 180,E1 13581.201,E2 13581.201} C_VEL
LIN {X 0,Y 280.926,Z 1034.054,A -85,B 0,C 180,E1 13577.461,E2 13577.461} C_VEL
LIN {X 0,Y 281.556,Z 1027.032,A -85,B 0,C 180,E1 13573.708,E2 13573.708} C_VEL
LIN {X 0,Y 283.018,Z 1018.457,A -85,B 0,C 180,E1 13570.175,E2 13570.175} C_VEL
LIN {X 0,Y 285.27,Z 1008.41,A -85,B 0,C 180,E1 13566.887,E2 13566.887} C_VEL
LIN {X 0,Y 288.186,Z 996.896,A -85,B 0,C 180,E1 13563.856,E2 13563.856} C_VEL
LIN {X 0,Y 291.625,Z 983.85,A -85,B 0,C 180,E1 13561.091,E2 13561.091} C_VEL
LIN {X 0,Y 295.353,Z 969.807,A -85,B 0,C 180,E1 13558.692,E2 13558.692} C_VEL
LIN {X 0,Y 299.266,Z 954.143,A -85,B 0,C 180,E1 13556.546,E2 13556.546} C_VEL
LIN {X 0,Y 302.882,Z 938.2,A -85,B 0,C 180,E1 13554.827,E2 13554.827} C_VEL
LIN {X 0,Y 306.149,Z 921.739,A -85,B 0,C 180,E1 13553.457,E2 13553.457} C_VEL
LIN {X 0,Y 309.031,Z 903.871,A -85,B 0,C 180,E1 13552.361,E2 13552.361} C_VEL
LIN {X 0,Y 311.084,Z 885.688,A -85,B 0,C 180,E1 13551.594,E2 13551.594} C_VEL
LIN {X 0,Y 312.306,Z 863.483,A -85,B 0,C 180,E1 13551.013,E2 13551.013} C_VEL
LIN {X 0,Y 317.928,Z 731.116,A -85,B 0,C 180,E1 13547.987,E2 13547.987} C_VEL
LIN {X 0,Y 315.393,Z 702.385,A -85,B 0,C 180,E1 13546.665,E2 13546.665} C_VEL
LIN {X 0,Y 314.727,Z 698.078,A -85,B 0,C 180,E1 13546.413,E2 13546.413} C_VEL
LIN {X 0,Y 313.89,Z 695.949,A -85,B 0,C 180,E1 13546.02,E2 13546.02} C_VEL
LIN {X 0,Y 310.31,Z 683.691,A -85,B 0,C 180,E1 13542.833,E2 13542.833} C_VEL
LIN {X 0,Y 306.273,Z 672.108,A -85,B 0,C 180,E1 13539.296,E2 13539.296} C_VEL
LIN {X 0,Y 302.483,Z 662.42,A -85,B 0,C 180,E1 13535.808,E2 13535.808} C_VEL
LIN {X 0,Y 299.558,Z 655.689,A -85,B 0,C 180,E1 13532.96,E2 13532.96} C_VEL
LIN {X 0,Y 297.653,Z 651.449,A -85,B 0,C 180,E1 13530.927,E2 13530.927} C_VEL
LIN {X 0,Y 296.274,Z 648.308,A -85,B 0,C 180,E1 13529.297,E2 13529.297} C_VEL
LIN {X 0,Y 294.367,Z 644.17,A -85,B 0,C 180,E1 13526.856,E2 13526.856} C_VEL
LIN {X 0,Y 292.424,Z 640.055,A -85,B 0,C 180,E1 13524.009,E2 13524.009} C_VEL
LIN {X 0,Y 290.143,Z 635.467,A -85,B 0,C 180,E1 13519.947,E2 13519.947} C_VEL
LIN {X 0,Y 287.814,Z 630.849,A -85,B 0,C 180,E1 13513.459,E2 13513.459} C_VEL
LIN {X 0,Y 286.884,Z 629.744,A -85,B 0,C 180,E1 13508.215,E2 13508.215} C_VEL
LIN {X 0,Y 287.319,Z 630.295,A -85,B 0,C 180,E1 13502.792,E2 13502.792} C_VEL
LIN {X 0,Y 287.895,Z 631.477,A -85,B 0,C 180,E1 13500,E2 13500} C_VEL
LIN {X 0,Y 289.977,Z 635.594,A -85,B 0,C 180,E1 13494.261,E2 13494.261} C_VEL
LIN {X 0,Y 291.953,Z 640.186,A -85,B 0,C 180,E1 13490.14,E2 13490.14} C_VEL
LIN {X 0,Y 293.804,Z 644.553,A -85,B 0,C 180,E1 13487.02,E2 13487.02} C_VEL
LIN {X 0,Y 295.572,Z 649,A -85,B 0,C 180,E1 13484.298,E2 13484.298} C_VEL
LIN {X 0,Y 297.955,Z 654.86,A -85,B 0,C 180,E1 13481.141,E2 13481.141} C_VEL
LIN {X 0,Y 301.054,Z 663.725,A -85,B 0,C 180,E1 13477.133,E2 13477.133} C_VEL
LIN {X 0,Y 303.992,Z 673.32,A -85,B 0,C 180,E1 13473.428,E2 13473.428} C_VEL
LIN {X 0,Y 306.706,Z 683.913,A -85,B 0,C 180,E1 13469.864,E2 13469.864} C_VEL
LIN {X 0,Y 308.612,Z 693.647,A -85,B 0,C 180,E1 13466.968,E2 13466.968} C_VEL
LIN {X 0,Y 305.905,Z 704.736,A -85,B 0,C 180,E1 13464.799,E2 13464.799} C_VEL
LIN {X 0,Y 307.837,Z 715.313,A -85,B 0,C 180,E1 13463.992,E2 13463.992} C_VEL
LIN {X 0,Y 312.833,Z 743.342,A -85,B 0,C 180,E1 13462.188,E2 13462.188} C_VEL
LIN {X 0,Y 314.215,Z 753.898,A -85,B 0,C 180,E1 13461.615,E2 13461.615} C_VEL
LIN {X 0,Y 309.888,Z 841.549,A -85,B 0,C 180,E1 13459.415,E2 13459.415} C_VEL
LIN {X 0,Y 308.562,Z 857.827,A -85,B 0,C 180,E1 13458.668,E2 13458.668} C_VEL
LIN {X 0,Y 306.689,Z 872.955,A -85,B 0,C 180,E1 13457.653,E2 13457.653} C_VEL
LIN {X 0,Y 304.216,Z 887.559,A -85,B 0,C 180,E1 13456.308,E2 13456.308} C_VEL
LIN {X 0,Y 301.401,Z 901.07,A -85,B 0,C 180,E1 13454.691,E2 13454.691} C_VEL
LIN {X 0,Y 298.32,Z 913.44,A -85,B 0,C 180,E1 13452.776,E2 13452.776} C_VEL
LIN {X 0,Y 295.176,Z 924.662,A -85,B 0,C 180,E1 13450.569,E2 13450.569} C_VEL
LIN {X 0,Y 292.043,Z 934.61,A -85,B 0,C 180,E1 13448.043,E2 13448.043} C_VEL
LIN {X 0,Y 289.182,Z 943.025,A -85,B 0,C 180,E1 13445.268,E2 13445.268} C_VEL
LIN {X 0,Y 286.706,Z 949.739,A -85,B 0,C 180,E1 13442.247,E2 13442.247} C_VEL
LIN {X 0,Y 284.875,Z 954.519,A -85,B 0,C 180,E1 13439.2,E2 13439.2} C_VEL
LIN {X 0,Y 283.538,Z 957.622,A -85,B 0,C 180,E1 13435.93,E2 13435.93} C_VEL
LIN {X 0,Y 282.778,Z 958.942,A -85,B 0,C 180,E1 13432.651,E2 13432.651} C_VEL
LIN {X 0,Y 282.476,Z 958.376,A -85,B 0,C 180,E1 13429.219,E2 13429.219} C_VEL
LIN {X 0,Y 282.623,Z 956.155,A -85,B 0,C 180,E1 13426.018,E2 13426.018} C_VEL
LIN {X 0,Y 283.19,Z 952.133,A -85,B 0,C 180,E1 13422.852,E2 13422.852} C_VEL
LIN {X 0,Y 284.256,Z 946.271,A -85,B 0,C 180,E1 13419.72,E2 13419.72} C_VEL
LIN {X 0,Y 285.732,Z 938.825,A -85,B 0,C 180,E1 13416.833,E2 13416.833} C_VEL
LIN {X 0,Y 287.559,Z 929.963,A -85,B 0,C 180,E1 13414.187,E2 13414.187} C_VEL
LIN {X 0,Y 289.803,Z 918.675,A -85,B 0,C 180,E1 13411.581,E2 13411.581} C_VEL
LIN {X 0,Y 291.976,Z 906.734,A -85,B 0,C 180,E1 13409.425,E2 13409.425} C_VEL
LIN {X 0,Y 294.244,Z 893.033,A -85,B 0,C 180,E1 13407.489,E2 13407.489} C_VEL
LIN {X 0,Y 296.228,Z 878.644,A -85,B 0,C 180,E1 13405.935,E2 13405.935} C_VEL
LIN {X 0,Y 297.886,Z 863.534,A -85,B 0,C 180,E1 13404.703,E2 13404.703} C_VEL
LIN {X 0,Y 299.155,Z 846.652,A -85,B 0,C 180,E1 13403.752,E2 13403.752} C_VEL
LIN {X 0,Y 299.846,Z 829.623,A -85,B 0,C 180,E1 13403.171,E2 13403.171} C_VEL
LIN {X 0,Y 302.692,Z 747.935,A -85,B 0,C 180,E1 13401.164,E2 13401.164} C_VEL
LIN {X 0,Y 296.261,Z 705.189,A -85,B 0,C 180,E1 13399.204,E2 13399.204} C_VEL
LIN {X 0,Y 300.704,Z 680.624,A -85,B 0,C 180,E1 13394.573,E2 13394.573} C_VEL
LIN {X 0,Y 297.101,Z 665.555,A -85,B 0,C 180,E1 13390.742,E2 13390.742} C_VEL
LIN {X 0,Y 293.242,Z 651.702,A -85,B 0,C 180,E1 13386.913,E2 13386.913} C_VEL
LIN {X 0,Y 289.477,Z 639.818,A -85,B 0,C 180,E1 13383.318,E2 13383.318} C_VEL
LIN {X 0,Y 285.004,Z 627.462,A -85,B 0,C 180,E1 13379.189,E2 13379.189} C_VEL
LIN {X 0,Y 282.431,Z 620.736,A -85,B 0,C 180,E1 13376.598,E2 13376.598} C_VEL
LIN {X 0,Y 282.421,Z 620.595,A -85,B 0,C 180,E1 13371.809,E2 13371.809} C_VEL
LIN {X 0,Y 282.419,Z 620.618,A -85,B 0,C 180,E1 13370.237,E2 13370.237} C_VEL
LIN {X 0,Y 281.607,Z 620.742,A -85,B 0,C 180,E1 13368.784,E2 13368.784} C_VEL
LIN {X 0,Y 278.155,Z 621.183,A -85,B 0,C 180,E1 13366.487,E2 13366.487} C_VEL
LIN {X 0,Y 274.842,Z 621.568,A -85,B 0,C 180,E1 13364.009,E2 13364.009} C_VEL
LIN {X 0,Y 274.469,Z 621.595,A -85,B 0,C 180,E1 13363.074,E2 13363.074} C_VEL
LIN {X 0,Y 274.461,Z 621.602,A -85,B 0,C 180,E1 13358.266,E2 13358.266} C_VEL
LIN {X 0,Y 274.473,Z 621.563,A -85,B 0,C 180,E1 13353.372,E2 13353.372} C_VEL
LIN {X 0,Y 274.48,Z 621.591,A -85,B 0,C 180,E1 13348.609,E2 13348.609} C_VEL
LIN {X 0,Y 274.454,Z 621.58,A -85,B 0,C 180,E1 13343.853,E2 13343.853} C_VEL
LIN {X 0,Y 274.456,Z 621.567,A -85,B 0,C 180,E1 13339.14,E2 13339.14} C_VEL
LIN {X 0,Y 274.486,Z 621.597,A -85,B 0,C 180,E1 13334.313,E2 13334.313} C_VEL
LIN {X 0,Y 274.454,Z 621.556,A -85,B 0,C 180,E1 13329.648,E2 13329.648} C_VEL
LIN {X 0,Y 274.45,Z 621.608,A -85,B 0,C 180,E1 13324.807,E2 13324.807} C_VEL
LIN {X 0,Y 274.469,Z 621.556,A -85,B 0,C 180,E1 13320,E2 13320} C_VEL
LIN {X 0,Y 274.458,Z 621.594,A -85,B 0,C 180,E1 13315.194,E2 13315.194} C_VEL
LIN {X 0,Y 274.443,Z 621.587,A -85,B 0,C 180,E1 13310.564,E2 13310.564} C_VEL
LIN {X 0,Y 274.449,Z 621.572,A -85,B 0,C 180,E1 13305.718,E2 13305.718} C_VEL
LIN {X 0,Y 274.471,Z 621.592,A -85,B 0,C 180,E1 13301.082,E2 13301.082} C_VEL
LIN {X 0,Y 274.455,Z 621.612,A -85,B 0,C 180,E1 13296.376,E2 13296.376} C_VEL
LIN {X 0,Y 274.443,Z 621.612,A -85,B 0,C 180,E1 13291.494,E2 13291.494} C_VEL
LIN {X 0,Y 274.54,Z 621.995,A -85,B 0,C 180,E1 13290.69,E2 13290.69} C_VEL
LIN {X 0,Y 279.544,Z 633.829,A -85,B 0,C 180,E1 13286.577,E2 13286.577} C_VEL
LIN {X 0,Y 284.865,Z 646.977,A -85,B 0,C 180,E1 13282.612,E2 13282.612} C_VEL
LIN {X 0,Y 290.347,Z 662.223,A -85,B 0,C 180,E1 13278.61,E2 13278.61} C_VEL
LIN {X 0,Y 295.696,Z 678.838,A -85,B 0,C 180,E1 13274.758,E2 13274.758} C_VEL
LIN {X 0,Y 299.278,Z 691.44,A -85,B 0,C 180,E1 13272.126,E2 13272.126} C_VEL
LIN {X 0,Y 298.33,Z 696.696,A -85,B 0,C 180,E1 13271.455,E2 13271.455} C_VEL
LIN {X 0,Y 301.107,Z 733.398,A -85,B 0,C 180,E1 13270.117,E2 13270.117} C_VEL
LIN {X 0,Y 295.775,Z 882.627,A -85,B 0,C 180,E1 13266.661,E2 13266.661} C_VEL
LIN {X 0,Y 294.273,Z 900.939,A -85,B 0,C 180,E1 13265.912,E2 13265.912} C_VEL
LIN {X 0,Y 292.024,Z 919.093,A -85,B 0,C 180,E1 13264.816,E2 13264.816} C_VEL
LIN {X 0,Y 289.44,Z 935.845,A -85,B 0,C 180,E1 13263.435,E2 13263.435} C_VEL
LIN {X 0,Y 286.544,Z 952.344,A -85,B 0,C 180,E1 13261.667,E2 13261.667} C_VEL
LIN {X 0,Y 283.559,Z 967.654,A -85,B 0,C 180,E1 13259.582,E2 13259.582} C_VEL
LIN {X 0,Y 280.617,Z 982.043,A -85,B 0,C 180,E1 13257.135,E2 13257.135} C_VEL
LIN {X 0,Y 278.045,Z 994.944,A -85,B 0,C 180,E1 13254.428,E2 13254.428} C_VEL
LIN {X 0,Y 275.784,Z 1007.184,A -85,B 0,C 180,E1 13251.257,E2 13251.257} C_VEL
LIN {X 0,Y 274.254,Z 1017.153,A -85,B 0,C 180,E1 13248.053,E2 13248.053} C_VEL
LIN {X 0,Y 273.381,Z 1025.697,A -85,B 0,C 180,E1 13244.618,E2 13244.618} C_VEL
LIN {X 0,Y 273.158,Z 1032.69,A -85,B 0,C 180,E1 13240.973,E2 13240.973} C_VEL
LIN {X 0,Y 273.492,Z 1037.743,A -85,B 0,C 180,E1 13237.352,E2 13237.352} C_VEL
LIN {X 0,Y 273.976,Z 1040.85,A -85,B 0,C 180,E1 13233.976,E2 13233.976} C_VEL
LIN {X 0,Y 274.261,Z 1042.285,A -85,B 0,C 180,E1 13230.836,E2 13230.836} C_VEL
LIN {X 0,Y 274.089,Z 1042.33,A -85,B 0,C 180,E1 13227.701,E2 13227.701} C_VEL
LIN {X 0,Y 273.559,Z 1040.905,A -85,B 0,C 180,E1 13224.337,E2 13224.337} C_VEL
LIN {X 0,Y 273.036,Z 1037.769,A -85,B 0,C 180,E1 13220.728,E2 13220.728} C_VEL
LIN {X 0,Y 272.987,Z 1032.629,A -85,B 0,C 180,E1 13216.875,E2 13216.875} C_VEL
LIN {X 0,Y 273.754,Z 1025.539,A -85,B 0,C 180,E1 13213.011,E2 13213.011} C_VEL
LIN {X 0,Y 275.42,Z 1016.888,A -85,B 0,C 180,E1 13209.382,E2 13209.382} C_VEL
LIN {X 0,Y 277.902,Z 1006.743,A -85,B 0,C 180,E1 13206.011,E2 13206.011} C_VEL
LIN {X 0,Y 281.069,Z 995.082,A -85,B 0,C 180,E1 13202.913,E2 13202.913} C_VEL
LIN {X 0,Y 284.771,Z 981.945,A -85,B 0,C 180,E1 13200.094,E2 13200.094} C_VEL
LIN {X 0,Y 288.924,Z 967.168,A -85,B 0,C 180,E1 13197.562,E2 13197.562} C_VEL
LIN {X 0,Y 292.904,Z 951.922,A -85,B 0,C 180,E1 13195.483,E2 13195.483} C_VEL
LIN {X 0,Y 296.671,Z 935.955,A -85,B 0,C 180,E1 13193.772,E2 13193.772} C_VEL
LIN {X 0,Y 300.016,Z 919.492,A -85,B 0,C 180,E1 13192.419,E2 13192.419} C_VEL
LIN {X 0,Y 302.915,Z 901.81,A -85,B 0,C 180,E1 13191.357,E2 13191.357} C_VEL
LIN {X 0,Y 304.973,Z 883.576,A -85,B 0,C 180,E1 13190.6,E2 13190.6} C_VEL
LIN {X 0,Y 306.35,Z 857.603,A -85,B 0,C 180,E1 13189.941,E2 13189.941} C_VEL
LIN {X 0,Y 311.995,Z 732.182,A -85,B 0,C 180,E1 13187.026,E2 13187.026} C_VEL
LIN {X 0,Y 309.601,Z 703.677,A -85,B 0,C 180,E1 13185.67,E2 13185.67} C_VEL
LIN {X 0,Y 309.147,Z 701.835,A -85,B 0,C 180,E1 13185.525,E2 13185.525} C_VEL
LIN {X 0,Y 306.589,Z 696.796,A -85,B 0,C 180,E1 13184.783,E2 13184.783} C_VEL
LIN {X 0,Y 302.812,Z 684.41,A -85,B 0,C 180,E1 13181.329,E2 13181.329} C_VEL
LIN {X 0,Y 299.098,Z 674.062,A -85,B 0,C 180,E1 13177.915,E2 13177.915} C_VEL
LIN {X 0,Y 295.781,Z 665.48,A -85,B 0,C 180,E1 13174.604,E2 13174.604} C_VEL
LIN {X 0,Y 292.68,Z 658.189,A -85,B 0,C 180,E1 13171.283,E2 13171.283} C_VEL
LIN {X 0,Y 290.534,Z 653.579,A -85,B 0,C 180,E1 13168.803,E2 13168.803} C_VEL
LIN {X 0,Y 288.836,Z 649.819,A -85,B 0,C 180,E1 13166.523,E2 13166.523} C_VEL
LIN {X 0,Y 287.091,Z 645.972,A -85,B 0,C 180,E1 13163.828,E2 13163.828} C_VEL
LIN {X 0,Y 284.954,Z 641.548,A -85,B 0,C 180,E1 13159.886,E2 13159.886} C_VEL
LIN {X 0,Y 282.717,Z 637.017,A -85,B 0,C 180,E1 13153.452,E2 13153.452} C_VEL
LIN {X 0,Y 281.786,Z 635.902,A -85,B 0,C 180,E1 13148.365,E2 13148.365} C_VEL
LIN {X 0,Y 282.103,Z 636.349,A -85,B 0,C 180,E1 13143.047,E2 13143.047} C_VEL
LIN {X 0,Y 282.639,Z 637.43,A -85,B 0,C 180,E1 13140.202,E2 13140.202} C_VEL
LIN {X 0,Y 284.56,Z 641.504,A -85,B 0,C 180,E1 13134.353,E2 13134.353} C_VEL
LIN {X 0,Y 286.401,Z 645.849,A -85,B 0,C 180,E1 13130.353,E2 13130.353} C_VEL
LIN {X 0,Y 288.146,Z 650.178,A -85,B 0,C 180,E1 13127.168,E2 13127.168} C_VEL
LIN {X 0,Y 290.007,Z 654.985,A -85,B 0,C 180,E1 13124.194,E2 13124.194} C_VEL
LIN {X 0,Y 292.212,Z 660.813,A -85,B 0,C 180,E1 13121.03,E2 13121.03} C_VEL
LIN {X 0,Y 295.021,Z 669.008,A -85,B 0,C 180,E1 13117.271,E2 13117.271} C_VEL
LIN {X 0,Y 297.692,Z 678.072,A -85,B 0,C 180,E1 13113.682,E2 13113.682} C_VEL
LIN {X 0,Y 300.294,Z 688.699,A -85,B 0,C 180,E1 13110.037,E2 13110.037} C_VEL
LIN {X 0,Y 301.849,Z 696.801,A -85,B 0,C 180,E1 13107.546,E2 13107.546} C_VEL
LIN {X 0,Y 299.866,Z 704.715,A -85,B 0,C 180,E1 13105.989,E2 13105.989} C_VEL
LIN {X 0,Y 304.654,Z 730.841,A -85,B 0,C 180,E1 13104.065,E2 13104.065} C_VEL
LIN {X 0,Y 308.305,Z 754.741,A -85,B 0,C 180,E1 13102.599,E2 13102.599} C_VEL
LIN {X 0,Y 303.77,Z 842.083,A -85,B 0,C 180,E1 13100.373,E2 13100.373} C_VEL
LIN {X 0,Y 302.377,Z 858.388,A -85,B 0,C 180,E1 13099.617,E2 13099.617} C_VEL
LIN {X 0,Y 300.476,Z 873.085,A -85,B 0,C 180,E1 13098.622,E2 13098.622} C_VEL
LIN {X 0,Y 297.958,Z 887.496,A -85,B 0,C 180,E1 13097.299,E2 13097.299} C_VEL
LIN {X 0,Y 294.99,Z 901.186,A -85,B 0,C 180,E1 13095.658,E2 13095.658} C_VEL
LIN {X 0,Y 291.866,Z 913.33,A -85,B 0,C 180,E1 13093.789,E2 13093.789} C_VEL
LIN {X 0,Y 288.397,Z 925.104,A -85,B 0,C 180,E1 13091.467,E2 13091.467} C_VEL
LIN {X 0,Y 285.33,Z 934.481,A -85,B 0,C 180,E1 13089.106,E2 13089.106} C_VEL
LIN {X 0,Y 282.205,Z 943.137,A -85,B 0,C 180,E1 13086.276,E2 13086.276} C_VEL
LIN {X 0,Y 279.661,Z 949.758,A -85,B 0,C 180,E1 13083.407,E2 13083.407} C_VEL
LIN {X 0,Y 277.464,Z 955.065,A -85,B 0,C 180,E1 13080.133,E2 13080.133} C_VEL
LIN {X 0,Y 275.981,Z 958.393,A -85,B 0,C 180,E1 13076.927,E2 13076.927} C_VEL
LIN {X 0,Y 275.029,Z 960.003,A -85,B 0,C 180,E1 13073.572,E2 13073.572} C_VEL
LIN {X 0,Y 274.605,Z 959.928,A -85,B 0,C 180,E1 13070.237,E2 13070.237} C_VEL
LIN {X 0,Y 274.617,Z 958.127,A -85,B 0,C 180,E1 13066.934,E2 13066.934} C_VEL
LIN {X 0,Y 275.077,Z 954.645,A -85,B 0,C 180,E1 13063.666,E2 13063.666} C_VEL
LIN {X 0,Y 275.949,Z 949.738,A -85,B 0,C 180,E1 13060.649,E2 13060.649} C_VEL
LIN {X 0,Y 277.416,Z 942.509,A -85,B 0,C 180,E1 13057.455,E2 13057.455} C_VEL
LIN {X 0,Y 279.164,Z 934.317,A -85,B 0,C 180,E1 13054.725,E2 13054.725} C_VEL
LIN {X 0,Y 281.362,Z 923.939,A -85,B 0,C 180,E1 13052.036,E2 13052.036} C_VEL
LIN {X 0,Y 283.635,Z 912.386,A -85,B 0,C 180,E1 13049.697,E2 13049.697} C_VEL
LIN {X 0,Y 286.01,Z 899.185,A -85,B 0,C 180,E1 13047.595,E2 13047.595} C_VEL
LIN {X 0,Y 288.168,Z 885.299,A -85,B 0,C 180,E1 13045.895,E2 13045.895} C_VEL
LIN {X 0,Y 289.975,Z 871.166,A -85,B 0,C 180,E1 13044.558,E2 13044.558} C_VEL
LIN {X 0,Y 291.475,Z 855.168,A -85,B 0,C 180,E1 13043.463,E2 13043.463} C_VEL
LIN {X 0,Y 292.455,Z 838.899,A -85,B 0,C 180,E1 13042.72,E2 13042.72} C_VEL
LIN {X 0,Y 295.695,Z 748.948,A -85,B 0,C 180,E1 13040.428,E2 13040.428} C_VEL
LIN {X 0,Y 289.163,Z 705.2,A -85,B 0,C 180,E1 13038.38,E2 13038.38} C_VEL
LIN {X 0,Y 293.314,Z 683.007,A -85,B 0,C 180,E1 13034.112,E2 13034.112} C_VEL
LIN {X 0,Y 289.813,Z 668.166,A -85,B 0,C 180,E1 13030.238,E2 13030.238} C_VEL
LIN {X 0,Y 286.201,Z 655.094,A -85,B 0,C 180,E1 13026.53,E2 13026.53} C_VEL
LIN {X 0,Y 282.445,Z 643.242,A -85,B 0,C 180,E1 13022.828,E2 13022.828} C_VEL
LIN {X 0,Y 278.577,Z 632.237,A -85,B 0,C 180,E1 13019.073,E2 13019.073} C_VEL
LIN {X 0,Y 275.226,Z 624.092,A -85,B 0,C 180,E1 13015.925,E2 13015.925} C_VEL
LIN {X 0,Y 274.475,Z 621.654,A -85,B 0,C 180,E1 13014.86,E2 13014.86} C_VEL
LIN {X 0,Y 274.485,Z 621.608,A -85,B 0,C 180,E1 13010.125,E2 13010.125} C_VEL
LIN {X 0,Y 274.473,Z 621.59,A -85,B 0,C 180,E1 13005.264,E2 13005.264} C_VEL
LIN {X 0,Y 274.469,Z 621.595,A -85,B 0,C 180,E1 13003.074,E2 13003.074} C_VEL
LIN {X 0,Y 273.453,Z 621.703,A -85,B 0,C 180,E1 13001.467,E2 13001.467} C_VEL
LIN {X 0,Y 269.204,Z 622.253,A -85,B 0,C 180,E1 12998.647,E2 12998.647} C_VEL
LIN {X 0,Y 266.719,Z 622.562,A -85,B 0,C 180,E1 12996.423,E2 12996.423} C_VEL
LIN {X 0,Y 266.527,Z 622.57,A -85,B 0,C 180,E1 12995.701,E2 12995.701} C_VEL
LIN {X 0,Y 266.544,Z 622.589,A -85,B 0,C 180,E1 12990.791,E2 12990.791} C_VEL
LIN {X 0,Y 266.515,Z 622.545,A -85,B 0,C 180,E1 12986.037,E2 12986.037} C_VEL
LIN {X 0,Y 266.529,Z 622.593,A -85,B 0,C 180,E1 12981.109,E2 12981.109} C_VEL
LIN {X 0,Y 266.529,Z 622.549,A -85,B 0,C 180,E1 12976.183,E2 12976.183} C_VEL
LIN {X 0,Y 266.514,Z 622.574,A -85,B 0,C 180,E1 12971.469,E2 12971.469} C_VEL
LIN {X 0,Y 266.514,Z 622.565,A -85,B 0,C 180,E1 12966.679,E2 12966.679} C_VEL
LIN {X 0,Y 266.529,Z 622.552,A -85,B 0,C 180,E1 12961.935,E2 12961.935} C_VEL
LIN {X 0,Y 266.518,Z 622.594,A -85,B 0,C 180,E1 12957.205,E2 12957.205} C_VEL
LIN {X 0,Y 266.501,Z 622.553,A -85,B 0,C 180,E1 12952.238,E2 12952.238} C_VEL
LIN {X 0,Y 266.529,Z 622.575,A -85,B 0,C 180,E1 12947.433,E2 12947.433} C_VEL
LIN {X 0,Y 266.523,Z 622.596,A -85,B 0,C 180,E1 12942.761,E2 12942.761} C_VEL
LIN {X 0,Y 266.495,Z 622.576,A -85,B 0,C 180,E1 12937.93,E2 12937.93} C_VEL
LIN {X 0,Y 266.529,Z 622.628,A -85,B 0,C 180,E1 12933.005,E2 12933.005} C_VEL
LIN {X 0,Y 266.609,Z 623.091,A -85,B 0,C 180,E1 12932.53,E2 12932.53} C_VEL
LIN {X 0,Y 268.006,Z 626.36,A -85,B 0,C 180,E1 12931.232,E2 12931.232} C_VEL
LIN {X 0,Y 271.84,Z 635.195,A -85,B 0,C 180,E1 12928.019,E2 12928.019} C_VEL
LIN {X 0,Y 276.411,Z 646.495,A -85,B 0,C 180,E1 12924.382,E2 12924.382} C_VEL
LIN {X 0,Y 281.217,Z 659.264,A -85,B 0,C 180,E1 12920.738,E2 12920.738} C_VEL
LIN {X 0,Y 286.417,Z 674.866,A -85,B 0,C 180,E1 12916.826,E2 12916.826} C_VEL
LIN {X 0,Y 291.643,Z 692.235,A -85,B 0,C 180,E1 12912.95,E2 12912.95} C_VEL
LIN {X 0,Y 291.984,Z 693.472,A -85,B 0,C 180,E1 12912.69,E2 12912.69} C_VEL
LIN {X 0,Y 291.422,Z 696.836,A -85,B 0,C 180,E1 12912.27,E2 12912.27} C_VEL
LIN {X 0,Y 294.156,Z 734.132,A -85,B 0,C 180,E1 12910.874,E2 12910.874} C_VEL
LIN {X 0,Y 288.662,Z 881.998,A -85,B 0,C 180,E1 12907.386,E2 12907.386} C_VEL
LIN {X 0,Y 287.126,Z 900.26,A -85,B 0,C 180,E1 12906.625,E2 12906.625} C_VEL
LIN {X 0,Y 284.827,Z 918.257,A -85,B 0,C 180,E1 12905.52,E2 12905.52} C_VEL
LIN {X 0,Y 282.243,Z 934.512,A -85,B 0,C 180,E1 12904.16,E2 12904.16} C_VEL
LIN {X 0,Y 279.226,Z 951.097,A -85,B 0,C 180,E1 12902.355,E2 12902.355} C_VEL
LIN {X 0,Y 276.122,Z 966.488,A -85,B 0,C 180,E1 12900.221,E2 12900.221} C_VEL
LIN {X 0,Y 273.048,Z 980.906,A -85,B 0,C 180,E1 12897.714,E2 12897.714} C_VEL
LIN {X 0,Y 270.355,Z 993.825,A -85,B 0,C 180,E1 12894.937,E2 12894.937} C_VEL
LIN {X 0,Y 267.979,Z 1006.072,A -85,B 0,C 180,E1 12891.678,E2 12891.678} C_VEL
LIN {X 0,Y 266.366,Z 1016.045,A -85,B 0,C 180,E1 12888.38,E2 12888.38} C_VEL
LIN {X 0,Y 265.44,Z 1024.588,A -85,B 0,C 180,E1 12884.842,E2 12884.842} C_VEL
LIN {X 0,Y 265.201,Z 1031.571,A -85,B 0,C 180,E1 12881.086,E2 12881.086} C_VEL
LIN {X 0,Y 265.555,Z 1036.613,A -85,B 0,C 180,E1 12877.355,E2 12877.355} C_VEL
LIN {X 0,Y 266.073,Z 1039.698,A -85,B 0,C 180,E1 12873.879,E2 12873.879} C_VEL
LIN {X 0,Y 266.359,Z 1041.107,A -85,B 0,C 180,E1 12870.646,E2 12870.646} C_VEL
LIN {X 0,Y 266.134,Z 1041.095,A -85,B 0,C 180,E1 12867.416,E2 12867.416} C_VEL
LIN {X 0,Y 265.546,Z 1039.609,A -85,B 0,C 180,E1 12863.949,E2 12863.949} C_VEL
LIN {X 0,Y 265.024,Z 1036.41,A -85,B 0,C 180,E1 12860.226,E2 12860.226} C_VEL
LIN {X 0,Y 265.063,Z 1031.204,A -85,B 0,C 180,E1 12856.253,E2 12856.253} C_VEL
LIN {X 0,Y 265.989,Z 1024.043,A -85,B 0,C 180,E1 12852.273,E2 12852.273} C_VEL
LIN {X 0,Y 267.875,Z 1015.318,A -85,B 0,C 180,E1 12848.544,E2 12848.544} C_VEL
LIN {X 0,Y 270.601,Z 1005.076,A -85,B 0,C 180,E1 12845.088,E2 12845.088} C_VEL
LIN {X 0,Y 274.035,Z 993.346,A -85,B 0,C 180,E1 12841.922,E2 12841.922} C_VEL
LIN {X 0,Y 278.025,Z 980.089,A -85,B 0,C 180,E1 12839.052,E2 12839.052} C_VEL
LIN {X 0,Y 282.255,Z 965.774,A -85,B 0,C 180,E1 12836.575,E2 12836.575} C_VEL
LIN {X 0,Y 286.453,Z 950.448,A -85,B 0,C 180,E1 12834.468,E2 12834.468} C_VEL
LIN {X 0,Y 290.249,Z 935.018,A -85,B 0,C 180,E1 12832.802,E2 12832.802} C_VEL
LIN {X 0,Y 293.668,Z 918.891,A -85,B 0,C 180,E1 12831.46,E2 12831.46} C_VEL
LIN {X 0,Y 296.713,Z 901.076,A -85,B 0,C 180,E1 12830.377,E2 12830.377} C_VEL
LIN {X 0,Y 298.848,Z 882.925,A -85,B 0,C 180,E1 12829.613,E2 12829.613} C_VEL
LIN {X 0,Y 300.298,Z 857.055,A -85,B 0,C 180,E1 12828.943,E2 12828.943} C_VEL
LIN {X 0,Y 306.178,Z 733.17,A -85,B 0,C 180,E1 12826.018,E2 12826.018} C_VEL
LIN {X 0,Y 304.052,Z 706.393,A -85,B 0,C 180,E1 12824.71,E2 12824.71} C_VEL
LIN {X 0,Y 299.224,Z 697.471,A -85,B 0,C 180,E1 12823.367,E2 12823.367} C_VEL
LIN {X 0,Y 295.843,Z 686.722,A -85,B 0,C 180,E1 12820.199,E2 12820.199} C_VEL
LIN {X 0,Y 292.37,Z 676.882,A -85,B 0,C 180,E1 12816.76,E2 12816.76} C_VEL
LIN {X 0,Y 288.972,Z 668.116,A -85,B 0,C 180,E1 12813.14,E2 12813.14} C_VEL
LIN {X 0,Y 285.756,Z 660.494,A -85,B 0,C 180,E1 12809.331,E2 12809.331} C_VEL
LIN {X 0,Y 283.499,Z 655.737,A -85,B 0,C 180,E1 12806.384,E2 12806.384} C_VEL
LIN {X 0,Y 281.762,Z 651.889,A -85,B 0,C 180,E1 12803.64,E2 12803.64} C_VEL
LIN {X 0,Y 279.655,Z 647.492,A -85,B 0,C 180,E1 12799.638,E2 12799.638} C_VEL
LIN {X 0,Y 277.563,Z 643.118,A -85,B 0,C 180,E1 12793.329,E2 12793.329} C_VEL
LIN {X 0,Y 276.624,Z 642.027,A -85,B 0,C 180,E1 12788.103,E2 12788.103} C_VEL
LIN {X 0,Y 276.988,Z 642.518,A -85,B 0,C 180,E1 12782.689,E2 12782.689} C_VEL
LIN {X 0,Y 277.4,Z 643.639,A -85,B 0,C 180,E1 12780,E2 12780} C_VEL
LIN {X 0,Y 279.164,Z 647.431,A -85,B 0,C 180,E1 12774.45,E2 12774.45} C_VEL
LIN {X 0,Y 280.912,Z 651.805,A -85,B 0,C 180,E1 12770.369,E2 12770.369} C_VEL
LIN {X 0,Y 282.51,Z 655.819,A -85,B 0,C 180,E1 12767.324,E2 12767.324} C_VEL
LIN {X 0,Y 284.768,Z 661.589,A -85,B 0,C 180,E1 12763.686,E2 12763.686} C_VEL
LIN {X 0,Y 287.307,Z 668.935,A -85,B 0,C 180,E1 12759.846,E2 12759.846} C_VEL
LIN {X 0,Y 290.157,Z 678.139,A -85,B 0,C 180,E1 12755.791,E2 12755.791} C_VEL
LIN {X 0,Y 292.807,Z 688.545,A -85,B 0,C 180,E1 12751.885,E2 12751.885} C_VEL
LIN {X 0,Y 294.894,Z 698.822,A -85,B 0,C 180,E1 12748.523,E2 12748.523} C_VEL
LIN {X 0,Y 295.043,Z 700.328,A -85,B 0,C 180,E1 12748.084,E2 12748.084} C_VEL
LIN {X 0,Y 293.963,Z 704.481,A -85,B 0,C 180,E1 12747.261,E2 12747.261} C_VEL
LIN {X 0,Y 296.239,Z 717.23,A -85,B 0,C 180,E1 12746.216,E2 12746.216} C_VEL
LIN {X 0,Y 301.19,Z 746.421,A -85,B 0,C 180,E1 12744.19,E2 12744.19} C_VEL
LIN {X 0,Y 302.442,Z 756.651,A -85,B 0,C 180,E1 12743.597,E2 12743.597} C_VEL
LIN {X 0,Y 297.763,Z 842.85,A -85,B 0,C 180,E1 12741.369,E2 12741.369} C_VEL
LIN {X 0,Y 296.3,Z 859.143,A -85,B 0,C 180,E1 12740.602,E2 12740.602} C_VEL
LIN {X 0,Y 294.153,Z 874.841,A -85,B 0,C 180,E1 12739.516,E2 12739.516} C_VEL
LIN {X 0,Y 291.409,Z 889.478,A -85,B 0,C 180,E1 12738.121,E2 12738.121} C_VEL
LIN {X 0,Y 288.305,Z 902.936,A -85,B 0,C 180,E1 12736.454,E2 12736.454} C_VEL
LIN {X 0,Y 284.85,Z 915.445,A -85,B 0,C 180,E1 12734.448,E2 12734.448} C_VEL
LIN {X 0,Y 281.233,Z 927.006,A -85,B 0,C 180,E1 12732.08,E2 12732.08} C_VEL
LIN {X 0,Y 277.878,Z 936.542,A -85,B 0,C 180,E1 12729.559,E2 12729.559} C_VEL
LIN {X 0,Y 274.632,Z 945.017,A -85,B 0,C 180,E1 12726.661,E2 12726.661} C_VEL
LIN {X 0,Y 271.972,Z 951.422,A -85,B 0,C 180,E1 12723.719,E2 12723.719} C_VEL
LIN {X 0,Y 269.602,Z 956.773,A -85,B 0,C 180,E1 12720.217,E2 12720.217} C_VEL
LIN {X 0,Y 268.037,Z 959.907,A -85,B 0,C 180,E1 12716.831,E2 12716.831} C_VEL
LIN {X 0,Y 267.044,Z 961.36,A -85,B 0,C 180,E1 12713.15,E2 12713.15} C_VEL
LIN {X 0,Y 266.661,Z 960.898,A -85,B 0,C 180,E1 12709.722,E2 12709.722} C_VEL
LIN {X 0,Y 266.773,Z 958.617,A -85,B 0,C 180,E1 12706.102,E2 12706.102} C_VEL
LIN {X 0,Y 267.401,Z 954.419,A -85,B 0,C 180,E1 12702.595,E2 12702.595} C_VEL
LIN {X 0,Y 268.531,Z 948.686,A -85,B 0,C 180,E1 12699.347,E2 12699.347} C_VEL
LIN {X 0,Y 270.207,Z 940.905,A -85,B 0,C 180,E1 12696.16,E2 12696.16} C_VEL
LIN {X 0,Y 272.203,Z 932.012,A -85,B 0,C 180,E1 12693.369,E2 12693.369} C_VEL
LIN {X 0,Y 274.647,Z 920.71,A -85,B 0,C 180,E1 12690.625,E2 12690.625} C_VEL
LIN {X 0,Y 276.913,Z 909.315,A -85,B 0,C 180,E1 12688.448,E2 12688.448} C_VEL
LIN {X 0,Y 279.361,Z 895.712,A -85,B 0,C 180,E1 12686.409,E2 12686.409} C_VEL
LIN {X 0,Y 281.527,Z 881.537,A -85,B 0,C 180,E1 12684.771,E2 12684.771} C_VEL
LIN {X 0,Y 283.416,Z 865.953,A -85,B 0,C 180,E1 12683.416,E2 12683.416} C_VEL
LIN {X 0,Y 284.78,Z 849.795,A -85,B 0,C 180,E1 12682.434,E2 12682.434} C_VEL
LIN {X 0,Y 285.594,Z 833.053,A -85,B 0,C 180,E1 12681.794,E2 12681.794} C_VEL
LIN {X 0,Y 288.738,Z 750.067,A -85,B 0,C 180,E1 12679.67,E2 12679.67} C_VEL
LIN {X 0,Y 282.141,Z 704.807,A -85,B 0,C 180,E1 12677.463,E2 12677.463} C_VEL
LIN {X 0,Y 285.96,Z 685.484,A -85,B 0,C 180,E1 12673.652,E2 12673.652} C_VEL
LIN {X 0,Y 282.521,Z 670.708,A -85,B 0,C 180,E1 12669.695,E2 12669.695} C_VEL
LIN {X 0,Y 278.967,Z 657.708,A -85,B 0,C 180,E1 12665.883,E2 12665.883} C_VEL
LIN {X 0,Y 275.164,Z 645.7,A -85,B 0,C 180,E1 12662.006,E2 12662.006} C_VEL
LIN {X 0,Y 271.34,Z 635.109,A -85,B 0,C 180,E1 12658.2,E2 12658.2} C_VEL
LIN {X 0,Y 267.919,Z 626.213,A -85,B 0,C 180,E1 12654.658,E2 12654.658} C_VEL
LIN {X 0,Y 266.534,Z 622.642,A -85,B 0,C 180,E1 12653.039,E2 12653.039} C_VEL
LIN {X 0,Y 266.536,Z 622.57,A -85,B 0,C 180,E1 12648.107,E2 12648.107} C_VEL
LIN {X 0,Y 266.536,Z 622.587,A -85,B 0,C 180,E1 12643.301,E2 12643.301} C_VEL
LIN {X 0,Y 266.522,Z 622.583,A -85,B 0,C 180,E1 12638.518,E2 12638.518} C_VEL
LIN {X 0,Y 266.527,Z 622.57,A -85,B 0,C 180,E1 12635.701,E2 12635.701} C_VEL
LIN {X 0,Y 265.68,Z 622.662,A -85,B 0,C 180,E1 12634.161,E2 12634.161} C_VEL
LIN {X 0,Y 262.045,Z 623.135,A -85,B 0,C 180,E1 12631.608,E2 12631.608} C_VEL
LIN {X 0,Y 258.867,Z 623.542,A -85,B 0,C 180,E1 12628.97,E2 12628.97} C_VEL
LIN {X 0,Y 258.582,Z 623.556,A -85,B 0,C 180,E1 12628.101,E2 12628.101} C_VEL
LIN {X 0,Y 258.595,Z 623.571,A -85,B 0,C 180,E1 12623.039,E2 12623.039} C_VEL
LIN {X 0,Y 258.587,Z 623.53,A -85,B 0,C 180,E1 12618.253,E2 12618.253} C_VEL
LIN {X 0,Y 258.577,Z 623.587,A -85,B 0,C 180,E1 12613.416,E2 12613.416} C_VEL
LIN {X 0,Y 258.585,Z 623.528,A -85,B 0,C 180,E1 12608.45,E2 12608.45} C_VEL
LIN {X 0,Y 258.589,Z 623.576,A -85,B 0,C 180,E1 12603.769,E2 12603.769} C_VEL
LIN {X 0,Y 258.564,Z 623.547,A -85,B 0,C 180,E1 12598.893,E2 12598.893} C_VEL
LIN {X 0,Y 258.576,Z 623.547,A -85,B 0,C 180,E1 12594.008,E2 12594.008} C_VEL
LIN {X 0,Y 258.587,Z 623.589,A -85,B 0,C 180,E1 12589.153,E2 12589.153} C_VEL
LIN {X 0,Y 258.563,Z 623.556,A -85,B 0,C 180,E1 12584.295,E2 12584.295} C_VEL
LIN {X 0,Y 258.579,Z 623.553,A -85,B 0,C 180,E1 12579.352,E2 12579.352} C_VEL
LIN {X 0,Y 258.628,Z 623.842,A -85,B 0,C 180,E1 12574.711,E2 12574.711} C_VEL
LIN {X 0,Y 260.268,Z 627.605,A -85,B 0,C 180,E1 12573.044,E2 12573.044} C_VEL
LIN {X 0,Y 264.204,Z 636.666,A -85,B 0,C 180,E1 12569.529,E2 12569.529} C_VEL
LIN {X 0,Y 268.794,Z 647.912,A -85,B 0,C 180,E1 12565.67,E2 12565.67} C_VEL
LIN {X 0,Y 273.563,Z 660.659,A -85,B 0,C 180,E1 12561.853,E2 12561.853} C_VEL
LIN {X 0,Y 278.669,Z 675.763,A -85,B 0,C 180,E1 12557.86,E2 12557.86} C_VEL
LIN {X 0,Y 283.739,Z 692.796,A -85,B 0,C 180,E1 12553.894,E2 12553.894} C_VEL
LIN {X 0,Y 284.599,Z 696.3,A -85,B 0,C 180,E1 12553.174,E2 12553.174} C_VEL
LIN {X 0,Y 287.251,Z 734.999,A -85,B 0,C 180,E1 12551.662,E2 12551.662} C_VEL
LIN {X 0,Y 281.571,Z 881.362,A -85,B 0,C 180,E1 12548.138,E2 12548.138} C_VEL
LIN {X 0,Y 279.985,Z 899.679,A -85,B 0,C 180,E1 12547.356,E2 12547.356} C_VEL
LIN {X 0,Y 277.563,Z 917.956,A -85,B 0,C 180,E1 12546.205,E2 12546.205} C_VEL
LIN {X 0,Y 274.726,Z 935.101,A -85,B 0,C 180,E1 12544.722,E2 12544.722} C_VEL
LIN {X 0,Y 271.642,Z 951.324,A -85,B 0,C 180,E1 12542.883,E2 12542.883} C_VEL
LIN {X 0,Y 268.431,Z 966.552,A -85,B 0,C 180,E1 12540.685,E2 12540.685} C_VEL
LIN {X 0,Y 265.267,Z 980.826,A -85,B 0,C 180,E1 12538.11,E2 12538.11} C_VEL
LIN {X 0,Y 262.493,Z 993.6,A -85,B 0,C 180,E1 12535.254,E2 12535.254} C_VEL
LIN {X 0,Y 260.187,Z 1004.961,A -85,B 0,C 180,E1 12532.124,E2 12532.124} C_VEL
LIN {X 0,Y 258.427,Z 1015.347,A -85,B 0,C 180,E1 12528.576,E2 12528.576} C_VEL
LIN {X 0,Y 257.466,Z 1023.946,A -85,B 0,C 180,E1 12524.852,E2 12524.852} C_VEL
LIN {X 0,Y 257.254,Z 1030.781,A -85,B 0,C 180,E1 12520.979,E2 12520.979} C_VEL
LIN {X 0,Y 257.653,Z 1035.703,A -85,B 0,C 180,E1 12517.134,E2 12517.134} C_VEL
LIN {X 0,Y 258.205,Z 1038.659,A -85,B 0,C 180,E1 12513.553,E2 12513.553} C_VEL
LIN {X 0,Y 258.457,Z 1039.978,A -85,B 0,C 180,E1 12510.222,E2 12510.222} C_VEL
LIN {X 0,Y 258.136,Z 1039.814,A -85,B 0,C 180,E1 12506.892,E2 12506.892} C_VEL
LIN {X 0,Y 257.487,Z 1038.166,A -85,B 0,C 180,E1 12503.311,E2 12503.311} C_VEL
LIN {X 0,Y 257.001,Z 1034.805,A -85,B 0,C 180,E1 12499.464,E2 12499.464} C_VEL
LIN {X 0,Y 257.193,Z 1029.435,A -85,B 0,C 180,E1 12495.363,E2 12495.363} C_VEL
LIN {X 0,Y 258.361,Z 1022.114,A -85,B 0,C 180,E1 12491.264,E2 12491.264} C_VEL
LIN {X 0,Y 260.546,Z 1013.174,A -85,B 0,C 180,E1 12487.434,E2 12487.434} C_VEL
LIN {X 0,Y 263.601,Z 1002.707,A -85,B 0,C 180,E1 12483.897,E2 12483.897} C_VEL
LIN {X 0,Y 267.51,Z 990.291,A -85,B 0,C 180,E1 12480.56,E2 12480.56} C_VEL
LIN {X 0,Y 271.717,Z 977.188,A -85,B 0,C 180,E1 12477.753,E2 12477.753} C_VEL
LIN {X 0,Y 276.065,Z 963.137,A -85,B 0,C 180,E1 12475.346,E2 12475.346} C_VEL
LIN {X 0,Y 280.523,Z 947.402,A -85,B 0,C 180,E1 12473.217,E2 12473.217} C_VEL
LIN {X 0,Y 284.539,Z 931.458,A -85,B 0,C 180,E1 12471.54,E2 12471.54} C_VEL
LIN {X 0,Y 288.162,Z 914.594,A -85,B 0,C 180,E1 12470.195,E2 12470.195} C_VEL
LIN {X 0,Y 291.193,Z 896.633,A -85,B 0,C 180,E1 12469.16,E2 12469.16} C_VEL
LIN {X 0,Y 293.209,Z 878.401,A -85,B 0,C 180,E1 12468.443,E2 12468.443} C_VEL
LIN {X 0,Y 300.459,Z 734.167,A -85,B 0,C 180,E1 12464.97,E2 12464.97} C_VEL
LIN {X 0,Y 298.662,Z 710.216,A -85,B 0,C 180,E1 12463.768,E2 12463.768} C_VEL
LIN {X 0,Y 292.037,Z 698.448,A -85,B 0,C 180,E1 12461.884,E2 12461.884} C_VEL
LIN {X 0,Y 291.101,Z 695.876,A -85,B 0,C 180,E1 12461.218,E2 12461.218} C_VEL
LIN {X 0,Y 287.677,Z 685.446,A -85,B 0,C 180,E1 12457.713,E2 12457.713} C_VEL
LIN {X 0,Y 284.246,Z 676.169,A -85,B 0,C 180,E1 12454.007,E2 12454.007} C_VEL
LIN {X 0,Y 281.123,Z 668.594,A -85,B 0,C 180,E1 12450.334,E2 12450.334} C_VEL
LIN {X 0,Y 279.203,Z 664.146,A -85,B 0,C 180,E1 12447.806,E2 12447.806} C_VEL
LIN {X 0,Y 277.89,Z 661.222,A -85,B 0,C 180,E1 12445.906,E2 12445.906} C_VEL
LIN {X 0,Y 276.284,Z 657.587,A -85,B 0,C 180,E1 12443.232,E2 12443.232} C_VEL
LIN {X 0,Y 274.474,Z 653.582,A -85,B 0,C 180,E1 12439.581,E2 12439.581} C_VEL
LIN {X 0,Y 272.397,Z 649.201,A -85,B 0,C 180,E1 12433.154,E2 12433.154} C_VEL
LIN {X 0,Y 271.482,Z 648.158,A -85,B 0,C 180,E1 12428.045,E2 12428.045} C_VEL
LIN {X 0,Y 271.79,Z 648.597,A -85,B 0,C 180,E1 12422.741,E2 12422.741} C_VEL
LIN {X 0,Y 272.166,Z 649.611,A -85,B 0,C 180,E1 12420.21,E2 12420.21} C_VEL
LIN {X 0,Y 273.793,Z 653.38,A -85,B 0,C 180,E1 12414.551,E2 12414.551} C_VEL
LIN {X 0,Y 275.366,Z 657.467,A -85,B 0,C 180,E1 12410.596,E2 12410.596} C_VEL
LIN {X 0,Y 277.005,Z 661.807,A -85,B 0,C 180,E1 12407.28,E2 12407.28} C_VEL
LIN {X 0,Y 279.079,Z 667.222,A -85,B 0,C 180,E1 12403.772,E2 12403.772} C_VEL
LIN {X 0,Y 281.635,Z 675.07,A -85,B 0,C 180,E1 12399.639,E2 12399.639} C_VEL
LIN {X 0,Y 284.212,Z 684.045,A -85,B 0,C 180,E1 12395.666,E2 12395.666} C_VEL
LIN {X 0,Y 286.616,Z 693.925,A -85,B 0,C 180,E1 12391.904,E2 12391.904} C_VEL
LIN {X 0,Y 288.368,Z 703.558,A -85,B 0,C 180,E1 12388.719,E2 12388.719} C_VEL
LIN {X 0,Y 288.316,Z 705.844,A -85,B 0,C 180,E1 12388.422,E2 12388.422} C_VEL
LIN {X 0,Y 293.367,Z 734.045,A -85,B 0,C 180,E1 12386.207,E2 12386.207} C_VEL
LIN {X 0,Y 296.74,Z 757.366,A -85,B 0,C 180,E1 12384.663,E2 12384.663} C_VEL
LIN {X 0,Y 291.86,Z 843.456,A -85,B 0,C 180,E1 12382.411,E2 12382.411} C_VEL
LIN {X 0,Y 290.32,Z 859.834,A -85,B 0,C 180,E1 12381.632,E2 12381.632} C_VEL
LIN {X 0,Y 288.177,Z 874.911,A -85,B 0,C 180,E1 12380.584,E2 12380.584} C_VEL
LIN {X 0,Y 285.34,Z 889.579,A -85,B 0,C 180,E1 12379.19,E2 12379.19} C_VEL
LIN {X 0,Y 282.074,Z 903.183,A -85,B 0,C 180,E1 12377.501,E2 12377.501} C_VEL
LIN {X 0,Y 278.62,Z 915.287,A -85,B 0,C 180,E1 12375.572,E2 12375.572} C_VEL
LIN {X 0,Y 274.636,Z 927.406,A -85,B 0,C 180,E1 12373.086,E2 12373.086} C_VEL
LIN {X 0,Y 271.031,Z 937.187,A -85,B 0,C 180,E1 12370.487,E2 12370.487} C_VEL
LIN {X 0,Y 267.549,Z 945.733,A -85,B 0,C 180,E1 12367.528,E2 12367.528} C_VEL
LIN {X 0,Y 264.682,Z 952.263,A -85,B 0,C 180,E1 12364.516,E2 12364.516} C_VEL
LIN {X 0,Y 262.132,Z 957.618,A -85,B 0,C 180,E1 12360.993,E2 12360.993} C_VEL
LIN {X 0,Y 260.381,Z 960.946,A -85,B 0,C 180,E1 12357.495,E2 12357.495} C_VEL
LIN {X 0,Y 259.227,Z 962.524,A -85,B 0,C 180,E1 12353.649,E2 12353.649} C_VEL
LIN {X 0,Y 258.767,Z 962.204,A -85,B 0,C 180,E1 12350.114,E2 12350.114} C_VEL
LIN {X 0,Y 258.821,Z 960.022,A -85,B 0,C 180,E1 12346.38,E2 12346.38} C_VEL
LIN {X 0,Y 259.389,Z 956.211,A -85,B 0,C 180,E1 12342.918,E2 12342.918} C_VEL
LIN {X 0,Y 260.523,Z 950.518,A -85,B 0,C 180,E1 12339.479,E2 12339.479} C_VEL
LIN {X 0,Y 262.114,Z 943.417,A -85,B 0,C 180,E1 12336.351,E2 12336.351} C_VEL
LIN {X 0,Y 264.278,Z 934.135,A -85,B 0,C 180,E1 12333.253,E2 12333.253} C_VEL
LIN {X 0,Y 266.57,Z 924.073,A -85,B 0,C 180,E1 12330.644,E2 12330.644} C_VEL
LIN {X 0,Y 269.098,Z 912.101,A -85,B 0,C 180,E1 12328.195,E2 12328.195} C_VEL
LIN {X 0,Y 271.474,Z 899.692,A -85,B 0,C 180,E1 12326.198,E2 12326.198} C_VEL
LIN {X 0,Y 273.94,Z 884.83,A -85,B 0,C 180,E1 12324.344,E2 12324.344} C_VEL
LIN {X 0,Y 275.938,Z 869.602,A -85,B 0,C 180,E1 12322.923,E2 12322.923} C_VEL
LIN {X 0,Y 277.498,Z 853.343,A -85,B 0,C 180,E1 12321.83,E2 12321.83} C_VEL
LIN {X 0,Y 278.464,Z 836.125,A -85,B 0,C 180,E1 12321.105,E2 12321.105} C_VEL
LIN {X 0,Y 281.816,Z 751.059,A -85,B 0,C 180,E1 12318.87,E2 12318.87} C_VEL
LIN {X 0,Y 275.162,Z 704.796,A -85,B 0,C 180,E1 12316.552,E2 12316.552} C_VEL
LIN {X 0,Y 278.645,Z 688.102,A -85,B 0,C 180,E1 12313.21,E2 12313.21} C_VEL
LIN {X 0,Y 275.371,Z 673.771,A -85,B 0,C 180,E1 12309.266,E2 12309.266} C_VEL
LIN {X 0,Y 271.731,Z 660.324,A -85,B 0,C 180,E1 12305.198,E2 12305.198} C_VEL
LIN {X 0,Y 268.243,Z 649.245,A -85,B 0,C 180,E1 12301.502,E2 12301.502} C_VEL
LIN {X 0,Y 264.322,Z 637.947,A -85,B 0,C 180,E1 12297.316,E2 12297.316} C_VEL
LIN {X 0,Y 259.995,Z 627.21,A -85,B 0,C 180,E1 12292.756,E2 12292.756} C_VEL
